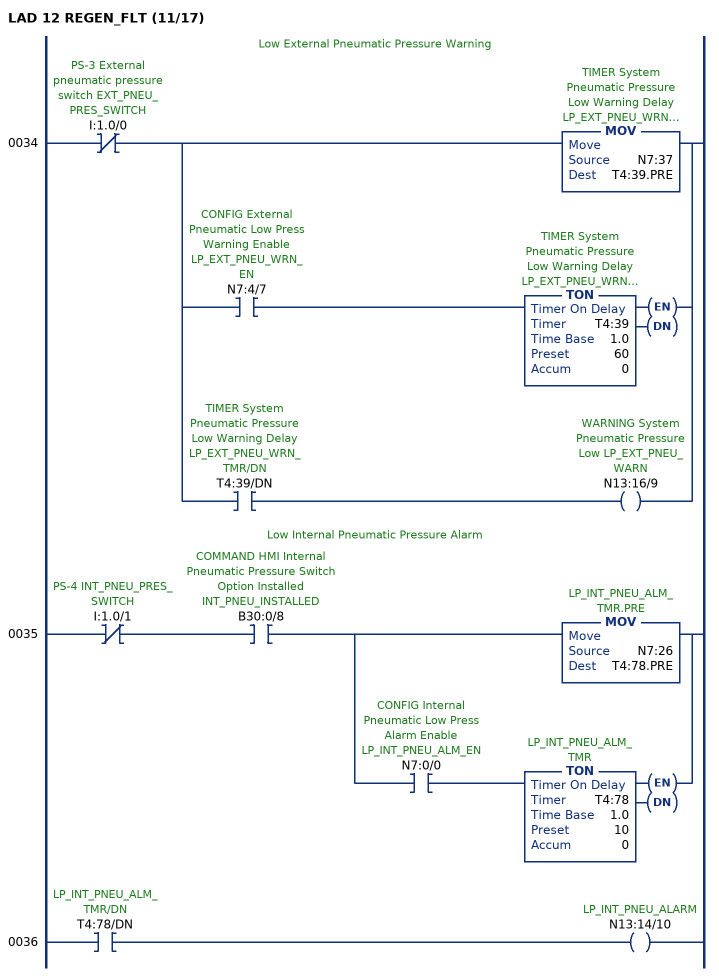
% Rung: 34 %
% Low External Pneumatic Pressure Warning %
SOR XIO I:1.0/0 BST MOV N7:37 T4:39.PRE NXB XIC N7:4/7 TON T4:39 1.0 60 0 NXB XIC T4:39/DN OTE N13:16/9 BND EOR
%   I:1.0/0  EXT_PNEU_PRES_SWITCH  "PS-3 External pneumatic pressure switch" %
%   N7:37  LP_EXT_PNEU_WRN_DLY  "CONFIG External Pneumatic Low Press Warning Delay" %
%   T4:39  LP_EXT_PNEU_WRN_TMR  "TIMER System Pneumatic Pressure Low Warning Delay" %
%   N7:4/7  LP_EXT_PNEU_WRN_EN  "CONFIG External Pneumatic Low Press Warning Enable" %
%   N13:16/9  LP_EXT_PNEU_WARN  "WARNING System Pneumatic Pressure Low" %
% Rung: 35 %
% Low Internal Pneumatic Pressure Alarm %
SOR XIO I:1.0/1 XIC B30:0/8 BST MOV N7:26 T4:78.PRE NXB XIC N7:0/0 TON T4:78 1.0 10 0 BND EOR
%   I:1.0/1  INT_PNEU_PRES_SWITCH  "PS-4" %
%   B30:0/8  INT_PNEU_INSTALLED  "COMMAND HMI Internal Pneumatic Pressure Switch Option Installed" %
%   N7:26  LP_INT_PNEU_ALM_DLY  "CONFIG Internal Pneumatic Low Press Alarm Delay" %
%   T4:78  LP_INT_PNEU_ALM_TMR %
%   N7:0/0  LP_INT_PNEU_ALM_EN  "CONFIG Internal Pneumatic Low Press Alarm Enable" %
% Rung: 36 %
SOR XIC T4:78/DN OTE N13:14/10 EOR
%   T4:78  LP_INT_PNEU_ALM_TMR %
%   N13:14/10  LP_INT_PNEU_ALARM %

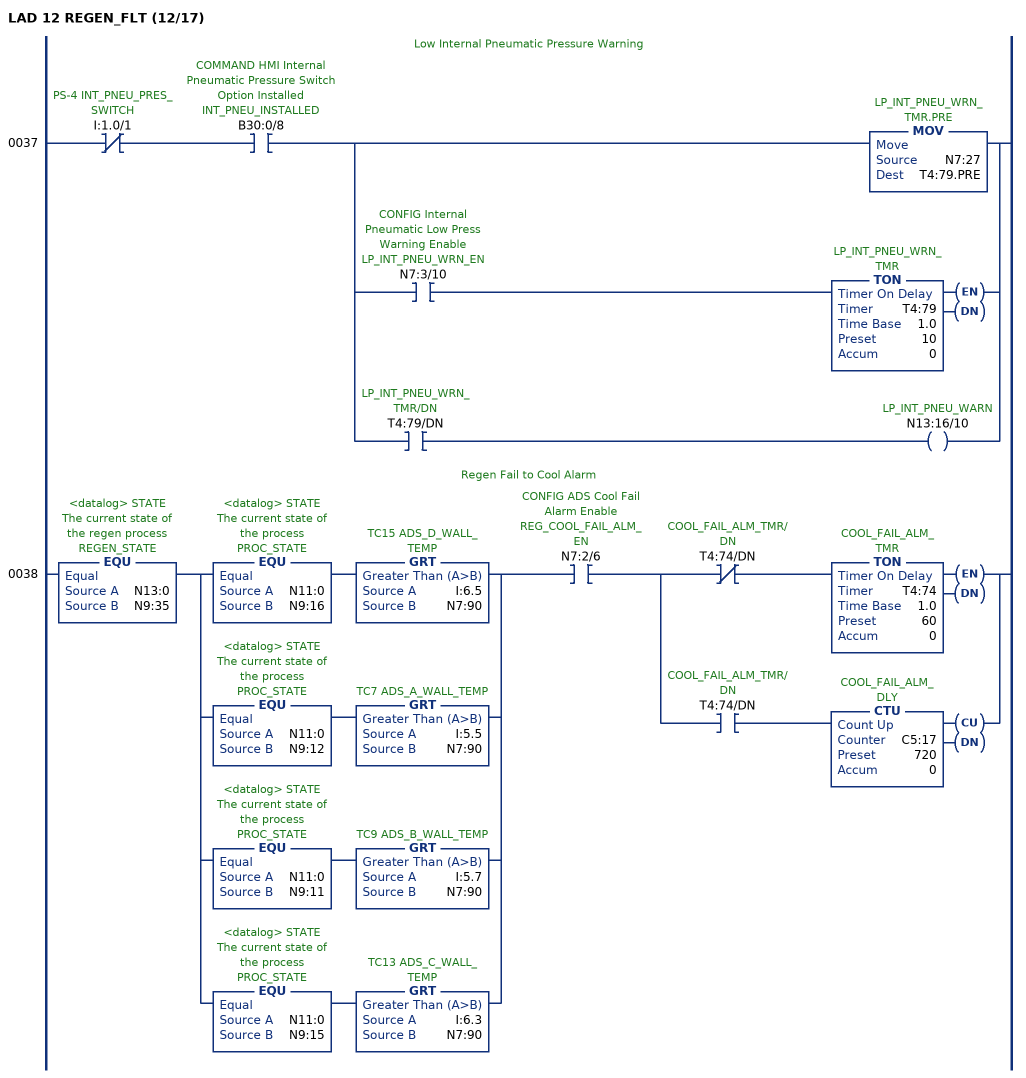
% Rung: 37 %
% Low Internal Pneumatic Pressure Warning %
SOR XIO I:1.0/1 XIC B30:0/8 BST MOV N7:27 T4:79.PRE NXB XIC N7:3/10 TON T4:79 1.0 10 0 NXB XIC T4:79/DN OTE N13:16/10 BND EOR
%   I:1.0/1  INT_PNEU_PRES_SWITCH  "PS-4" %
%   B30:0/8  INT_PNEU_INSTALLED  "COMMAND HMI Internal Pneumatic Pressure Switch Option Installed" %
%   N7:27  LP_INT_PNEU_WRN_DLY  "CONFIG Internal Pneumatic Low Press Warning Delay" %
%   T4:79  LP_INT_PNEU_WRN_TMR %
%   N7:3/10  LP_INT_PNEU_WRN_EN  "CONFIG Internal Pneumatic Low Press Warning Enable" %
%   N13:16/10  LP_INT_PNEU_WARN %
% Rung: 38 %
% Regen Fail to Cool Alarm %
SOR EQU N13:0 N9:35 BST EQU N11:0 N9:16 GRT I:6.5 N7:90 NXB EQU N11:0 N9:12 GRT I:5.5 N7:90 NXB EQU N11:0 N9:11 GRT I:5.7 N7:90 NXB EQU N11:0 N9:15 GRT I:6.3 N7:90 BND XIC N7:2/6 BST XIO T4:74/DN TON T4:74 1.0 60 0 NXB XIC T4:74/DN CTU C5:17 720 0 BND EOR
%   N13:0  REGEN_STATE  "<datalog> STATE The current state of the regen process" %
%   N9:35  REGEN_COOL_WALL  "STATE Regen Cool wall" %
%   N11:0  PROC_STATE  "<datalog> STATE The current state of the process" %
%   N9:16  PROC_REGEN_D  "STATE Process Regen D" %
%   I:6.5  ADS_D_WALL_TEMP  "TC15" %
%   N7:90  REG_COOL_FAIL_ALM_SP  "CONFIG ADS Cool Fail Alarm Setpoint" %
%   N9:12  PROC_REGEN_A  "STATE Process Regen A" %
%   I:5.5  ADS_A_WALL_TEMP  "TC7" %
%   N9:11  PROC_REGEN_B  "STATE Process Regen B" %
%   I:5.7  ADS_B_WALL_TEMP  "TC9" %
%   N9:15  PROC_REGEN_C  "STATE Process Regen C" %
%   I:6.3  ADS_C_WALL_TEMP  "TC13" %
%   N7:2/6  REG_COOL_FAIL_ALM_EN  "CONFIG ADS Cool Fail Alarm Enable" %
%   T4:74  COOL_FAIL_ALM_TMR %
%   C5:17  COOL_FAIL_ALM_DLY %

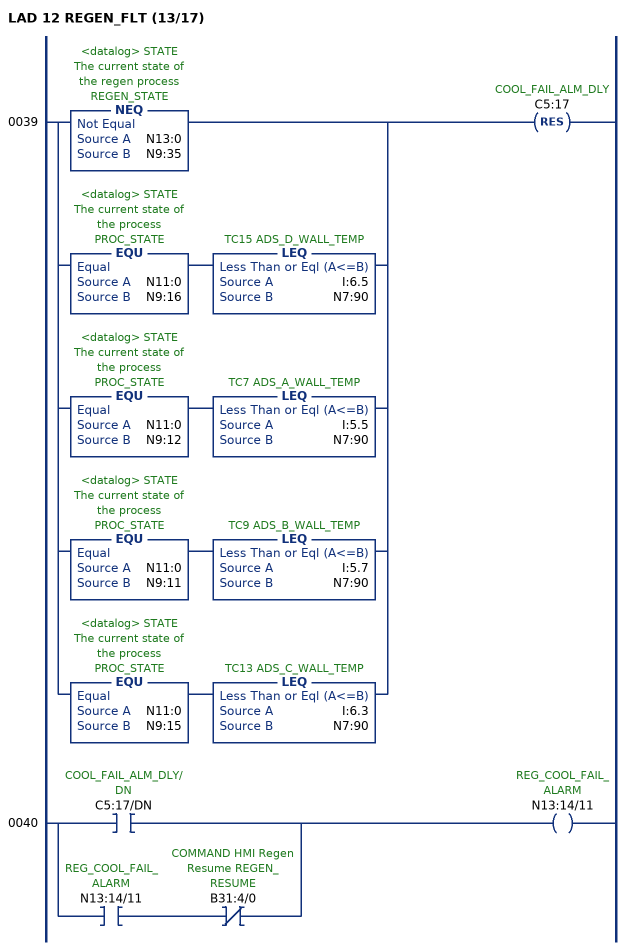
% Rung: 39 %
SOR BST NEQ N13:0 N9:35 NXB EQU N11:0 N9:16 LEQ I:6.5 N7:90 NXB EQU N11:0 N9:12 LEQ I:5.5 N7:90 NXB EQU N11:0 N9:11 LEQ I:5.7 N7:90 NXB EQU N11:0 N9:15 LEQ I:6.3 N7:90 BND RES C5:17 EOR
%   N13:0  REGEN_STATE  "<datalog> STATE The current state of the regen process" %
%   N9:35  REGEN_COOL_WALL  "STATE Regen Cool wall" %
%   N11:0  PROC_STATE  "<datalog> STATE The current state of the process" %
%   N9:16  PROC_REGEN_D  "STATE Process Regen D" %
%   I:6.5  ADS_D_WALL_TEMP  "TC15" %
%   N7:90  REG_COOL_FAIL_ALM_SP  "CONFIG ADS Cool Fail Alarm Setpoint" %
%   N9:12  PROC_REGEN_A  "STATE Process Regen A" %
%   I:5.5  ADS_A_WALL_TEMP  "TC7" %
%   N9:11  PROC_REGEN_B  "STATE Process Regen B" %
%   I:5.7  ADS_B_WALL_TEMP  "TC9" %
%   N9:15  PROC_REGEN_C  "STATE Process Regen C" %
%   I:6.3  ADS_C_WALL_TEMP  "TC13" %
%   C5:17  COOL_FAIL_ALM_DLY %
% Rung: 40 %
SOR BST XIC C5:17/DN NXB XIC N13:14/11 XIO B31:4/0 BND OTE N13:14/11 EOR
%   C5:17  COOL_FAIL_ALM_DLY %
%   N13:14/11  REG_COOL_FAIL_ALARM %
%   B31:4/0  REGEN_RESUME  "COMMAND HMI Regen Resume" %

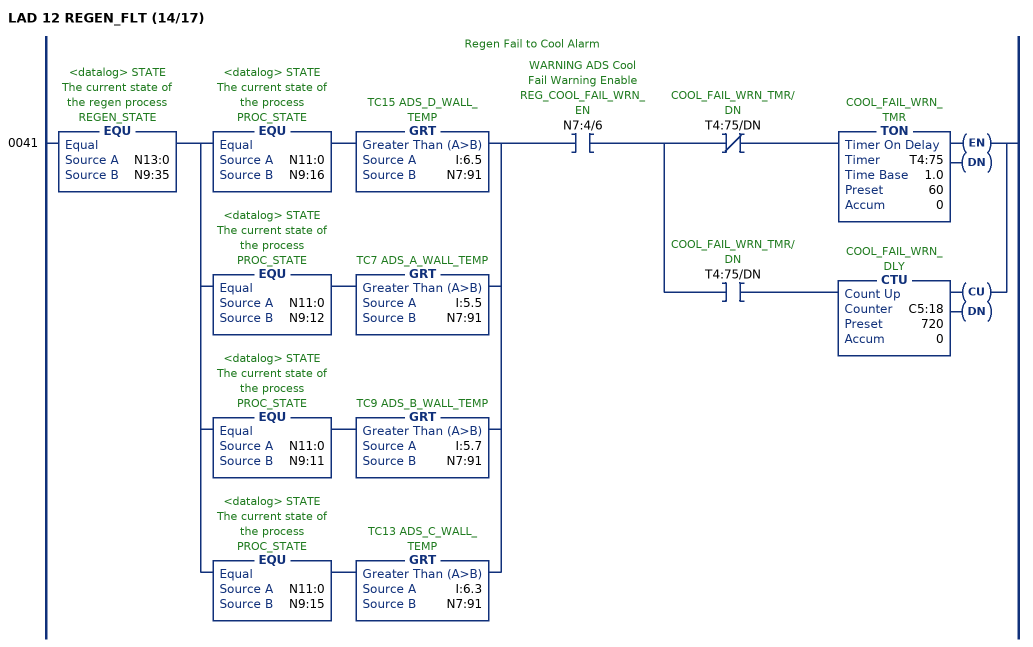
% Rung: 41 %
% Regen Fail to Cool Alarm %
SOR EQU N13:0 N9:35 BST EQU N11:0 N9:16 GRT I:6.5 N7:91 NXB EQU N11:0 N9:12 GRT I:5.5 N7:91 NXB EQU N11:0 N9:11 GRT I:5.7 N7:91 NXB EQU N11:0 N9:15 GRT I:6.3 N7:91 BND XIC N7:4/6 BST XIO T4:75/DN TON T4:75 1.0 60 0 NXB XIC T4:75/DN CTU C5:18 720 0 BND EOR
%   N13:0  REGEN_STATE  "<datalog> STATE The current state of the regen process" %
%   N9:35  REGEN_COOL_WALL  "STATE Regen Cool wall" %
%   N11:0  PROC_STATE  "<datalog> STATE The current state of the process" %
%   N9:16  PROC_REGEN_D  "STATE Process Regen D" %
%   I:6.5  ADS_D_WALL_TEMP  "TC15" %
%   N7:91  REG_COOL_FAIL_WRN_SP  "CONFIG ADS Cool Fail Warning Setpoint" %
%   N9:12  PROC_REGEN_A  "STATE Process Regen A" %
%   I:5.5  ADS_A_WALL_TEMP  "TC7" %
%   N9:11  PROC_REGEN_B  "STATE Process Regen B" %
%   I:5.7  ADS_B_WALL_TEMP  "TC9" %
%   N9:15  PROC_REGEN_C  "STATE Process Regen C" %
%   I:6.3  ADS_C_WALL_TEMP  "TC13" %
%   N7:4/6  REG_COOL_FAIL_WRN_EN  "WARNING ADS Cool Fail Warning Enable" %
%   T4:75  COOL_FAIL_WRN_TMR %
%   C5:18  COOL_FAIL_WRN_DLY %

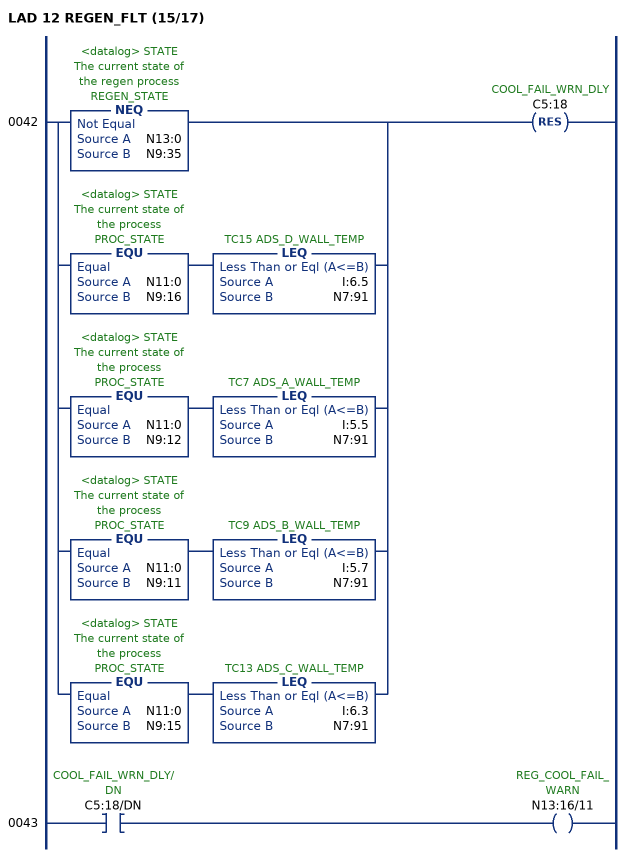
% Rung: 42 %
SOR BST NEQ N13:0 N9:35 NXB EQU N11:0 N9:16 LEQ I:6.5 N7:91 NXB EQU N11:0 N9:12 LEQ I:5.5 N7:91 NXB EQU N11:0 N9:11 LEQ I:5.7 N7:91 NXB EQU N11:0 N9:15 LEQ I:6.3 N7:91 BND RES C5:18 EOR
%   N13:0  REGEN_STATE  "<datalog> STATE The current state of the regen process" %
%   N9:35  REGEN_COOL_WALL  "STATE Regen Cool wall" %
%   N11:0  PROC_STATE  "<datalog> STATE The current state of the process" %
%   N9:16  PROC_REGEN_D  "STATE Process Regen D" %
%   I:6.5  ADS_D_WALL_TEMP  "TC15" %
%   N7:91  REG_COOL_FAIL_WRN_SP  "CONFIG ADS Cool Fail Warning Setpoint" %
%   N9:12  PROC_REGEN_A  "STATE Process Regen A" %
%   I:5.5  ADS_A_WALL_TEMP  "TC7" %
%   N9:11  PROC_REGEN_B  "STATE Process Regen B" %
%   I:5.7  ADS_B_WALL_TEMP  "TC9" %
%   N9:15  PROC_REGEN_C  "STATE Process Regen C" %
%   I:6.3  ADS_C_WALL_TEMP  "TC13" %
%   C5:18  COOL_FAIL_WRN_DLY %
% Rung: 43 %
SOR XIC C5:18/DN OTE N13:16/11 EOR
%   C5:18  COOL_FAIL_WRN_DLY %
%   N13:16/11  REG_COOL_FAIL_WARN %

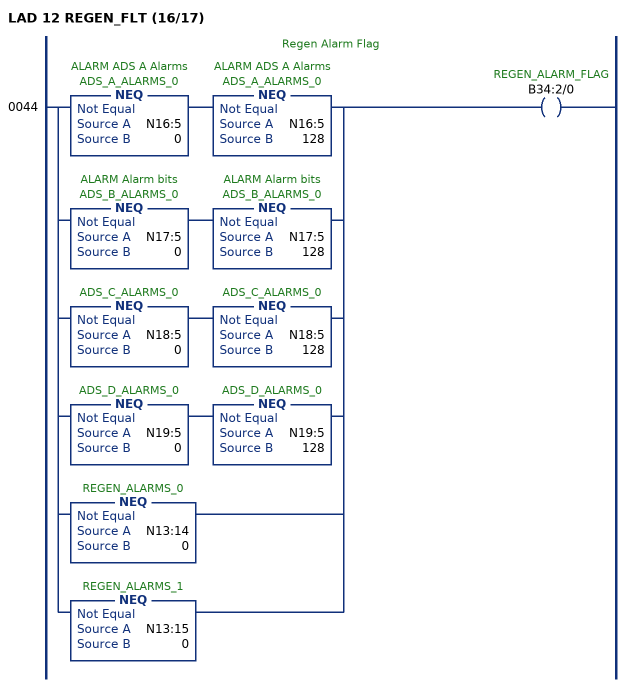
% Rung: 44 %
% Regen Alarm Flag %
SOR BST NEQ N16:5 0 NEQ N16:5 128 NXB NEQ N17:5 0 NEQ N17:5 128 NXB NEQ N18:5 0 NEQ N18:5 128 NXB NEQ N19:5 0 NEQ N19:5 128 NXB NEQ N13:14 0 NXB NEQ N13:15 0 BND OTE B34:2/0 EOR
%   N16:5  ADS_A_ALARMS_0  "ALARM ADS A Alarms" %
%   N17:5  ADS_B_ALARMS_0  "ALARM Alarm bits" %
%   N18:5  ADS_C_ALARMS_0 %
%   N19:5  ADS_D_ALARMS_0 %
%   N13:14  REGEN_ALARMS_0 %
%   N13:15  REGEN_ALARMS_1 %
%   B34:2/0  REGEN_ALARM_FLAG %

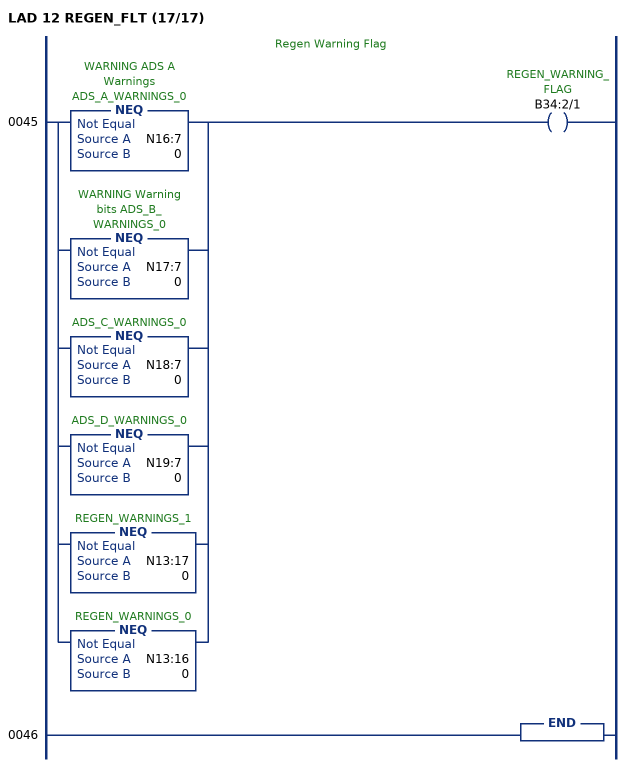
% Rung: 45 %
% Regen Warning Flag %
SOR BST NEQ N16:7 0 NXB NEQ N17:7 0 NXB NEQ N18:7 0 NXB NEQ N19:7 0 NXB NEQ N13:17 0 NXB NEQ N13:16 0 BND OTE B34:2/1 EOR
%   N16:7  ADS_A_WARNINGS_0  "WARNING ADS A Warnings" %
%   N17:7  ADS_B_WARNINGS_0  "WARNING Warning bits" %
%   N18:7  ADS_C_WARNINGS_0 %
%   N19:7  ADS_D_WARNINGS_0 %
%   N13:17  REGEN_WARNINGS_1 %
%   N13:16  REGEN_WARNINGS_0 %
%   B34:2/1  REGEN_WARNING_FLAG %
% Rung: 46 %
SOR END EOR

LADDER 17 "BYPASS"    % Controls the bypass %
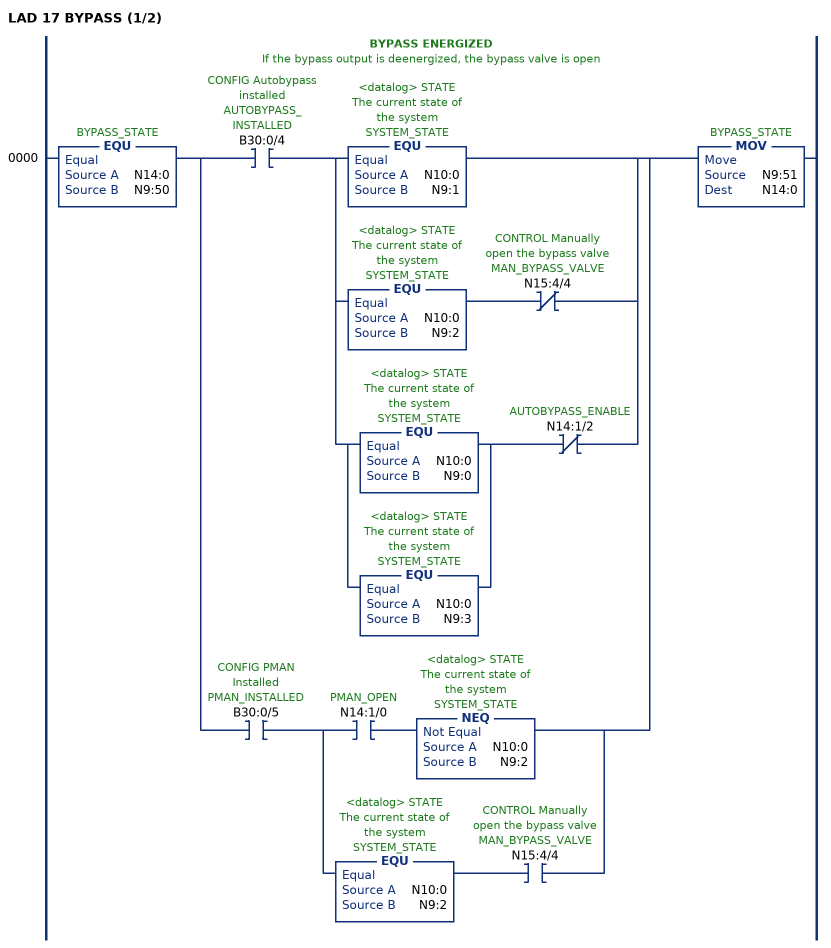
% Rung: 0 %
% TITLE: BYPASS ENERGIZED %
% If the bypass output is deenergized, the bypass valve is open %
SOR EQU N14:0 N9:50 BST XIC B30:0/4 BST EQU N10:0 N9:1 NXB EQU N10:0 N9:2 XIO N15:4/4 NXB BST EQU N10:0 N9:0 NXB EQU N10:0 N9:3 BND XIO N14:1/2 BND NXB XIC B30:0/5 BST XIC N14:1/0 NEQ N10:0 N9:2 NXB EQU N10:0 N9:2 XIC N15:4/4 BND BND MOV N9:51 N14:0 EOR
%   N14:0  BYPASS_STATE %
%   N9:50  BYPASS_DEENERGIZED  "STATE Bypass Deenergized" %
%   B30:0/4  AUTOBYPASS_INSTALLED  "CONFIG Autobypass installed" %
%   N10:0  SYSTEM_STATE  "<datalog> STATE The current state of the system" %
%   N9:1  SYSTEM_PROCESS  "STATE System Process" %
%   N9:2  SYSTEM_MANUAL  "STATE System Manual" %
%   N15:4/4  MAN_BYPASS_VALVE  "CONTROL Manually open the bypass valve" %
%   N9:0  SYSTEM_STANDBY  "STATE System Standby" %
%   N9:3  SYSTEM_ALARM  "STATE System Alarm" %
%   N14:1/2  AUTOBYPASS_ENABLE %
%   B30:0/5  PMAN_INSTALLED  "CONFIG PMAN Installed" %
%   N14:1/0  PMAN_OPEN %
%   N9:51  BYPASS_ENERGIZED  "STATE Bypass Energized" %

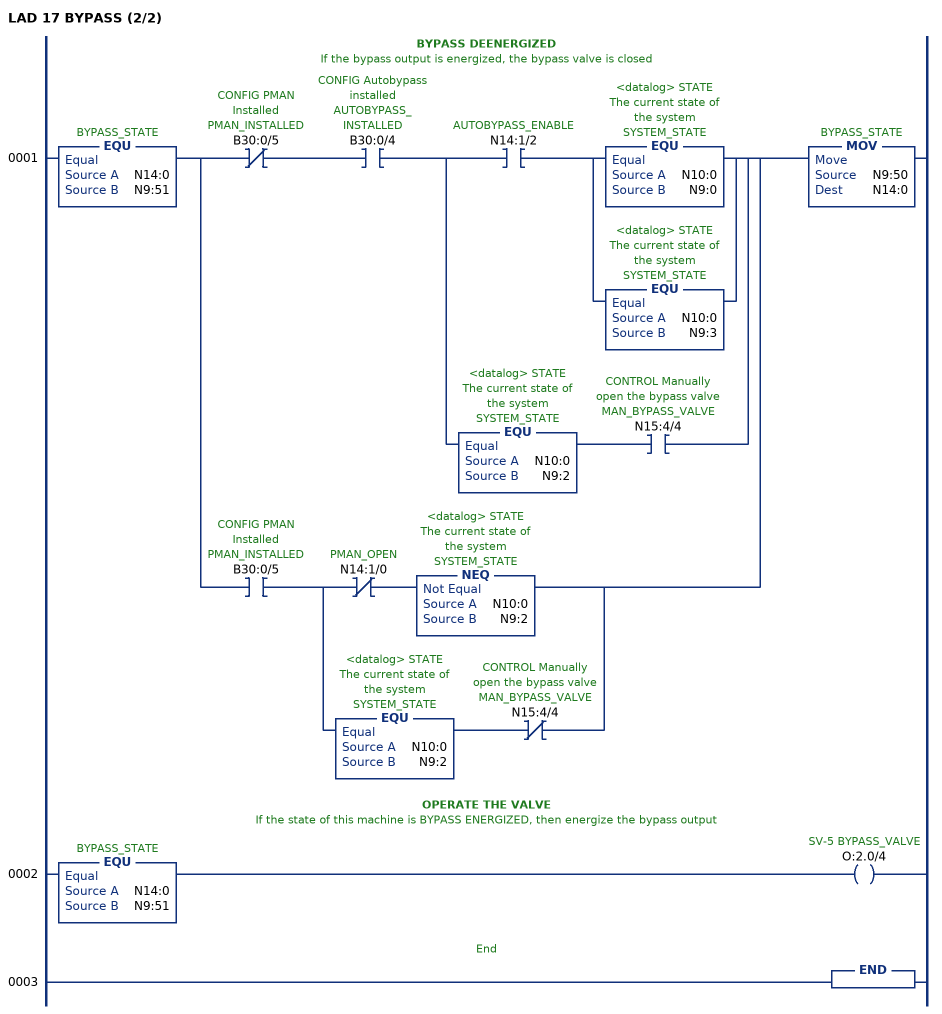
% Rung: 1 %
% TITLE: BYPASS DEENERGIZED %
% If the bypass output is energized, the bypass valve is closed %
SOR EQU N14:0 N9:51 BST XIO B30:0/5 XIC B30:0/4 BST XIC N14:1/2 BST EQU N10:0 N9:0 NXB EQU N10:0 N9:3 BND NXB EQU N10:0 N9:2 XIC N15:4/4 BND NXB XIC B30:0/5 BST XIO N14:1/0 NEQ N10:0 N9:2 NXB EQU N10:0 N9:2 XIO N15:4/4 BND BND MOV N9:50 N14:0 EOR
%   N14:0  BYPASS_STATE %
%   N9:51  BYPASS_ENERGIZED  "STATE Bypass Energized" %
%   B30:0/5  PMAN_INSTALLED  "CONFIG PMAN Installed" %
%   B30:0/4  AUTOBYPASS_INSTALLED  "CONFIG Autobypass installed" %
%   N14:1/2  AUTOBYPASS_ENABLE %
%   N10:0  SYSTEM_STATE  "<datalog> STATE The current state of the system" %
%   N9:0  SYSTEM_STANDBY  "STATE System Standby" %
%   N9:3  SYSTEM_ALARM  "STATE System Alarm" %
%   N9:2  SYSTEM_MANUAL  "STATE System Manual" %
%   N15:4/4  MAN_BYPASS_VALVE  "CONTROL Manually open the bypass valve" %
%   N14:1/0  PMAN_OPEN %
%   N9:50  BYPASS_DEENERGIZED  "STATE Bypass Deenergized" %
% Rung: 2 %
% TITLE: OPERATE THE VALVE %
% If the state of this machine is BYPASS ENERGIZED, then energize the bypass output %
SOR EQU N14:0 N9:51 OTE O:2.0/4 EOR
%   N14:0  BYPASS_STATE %
%   N9:51  BYPASS_ENERGIZED  "STATE Bypass Energized" %
%   O:2.0/4  BYPASS_VALVE  "SV-5" %
% Rung: 3 %
% End %
SOR END EOR

LADDER 18 "MIX PANEL"
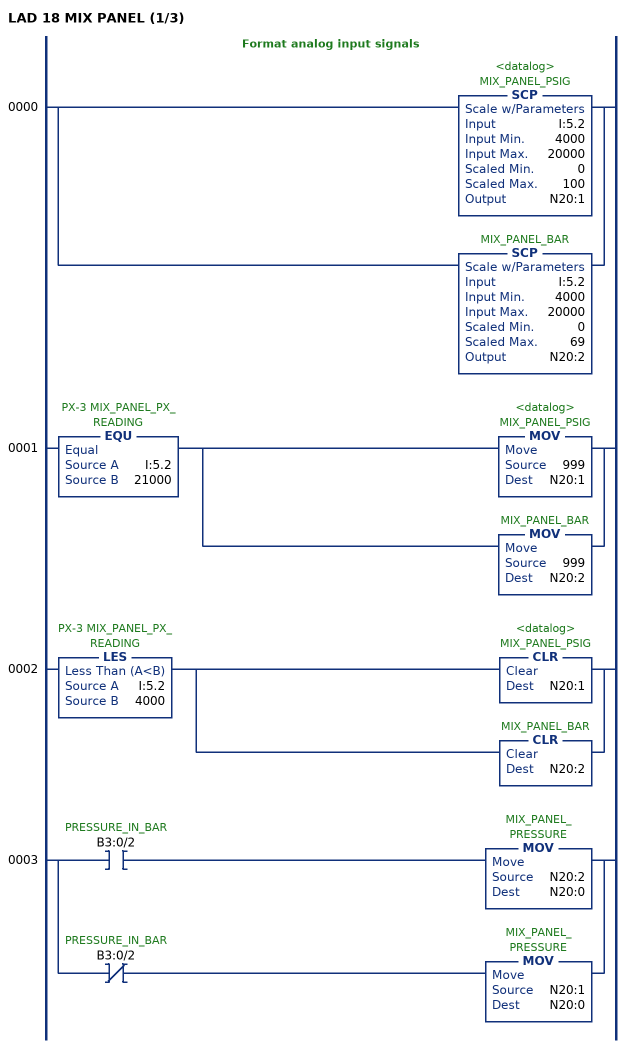
% Rung: 0 %
% TITLE: Format analog input signals %
SOR BST SCP I:5.2 4000 20000 0 100 N20:1 NXB SCP I:5.2 4000 20000 0 69 N20:2 BND EOR
%   I:5.2  MIX_PANEL_PX_READING  "PX-3" %
%   N20:1  MIX_PANEL_PSIG  "<datalog>" %
%   N20:2  MIX_PANEL_BAR %
% Rung: 1 %
SOR EQU I:5.2 21000 BST MOV 999 N20:1 NXB MOV 999 N20:2 BND EOR
%   I:5.2  MIX_PANEL_PX_READING  "PX-3" %
%   N20:1  MIX_PANEL_PSIG  "<datalog>" %
%   N20:2  MIX_PANEL_BAR %
% Rung: 2 %
SOR LES I:5.2 4000 BST CLR N20:1 NXB CLR N20:2 BND EOR
%   I:5.2  MIX_PANEL_PX_READING  "PX-3" %
%   N20:1  MIX_PANEL_PSIG  "<datalog>" %
%   N20:2  MIX_PANEL_BAR %
% Rung: 3 %
SOR BST XIC B3:0/2 MOV N20:2 N20:0 NXB XIO B3:0/2 MOV N20:1 N20:0 BND EOR
%   B3:0/2  PRESSURE_IN_BAR %
%   N20:2  MIX_PANEL_BAR %
%   N20:0  MIX_PANEL_PRESSURE %
%   N20:1  MIX_PANEL_PSIG  "<datalog>" %

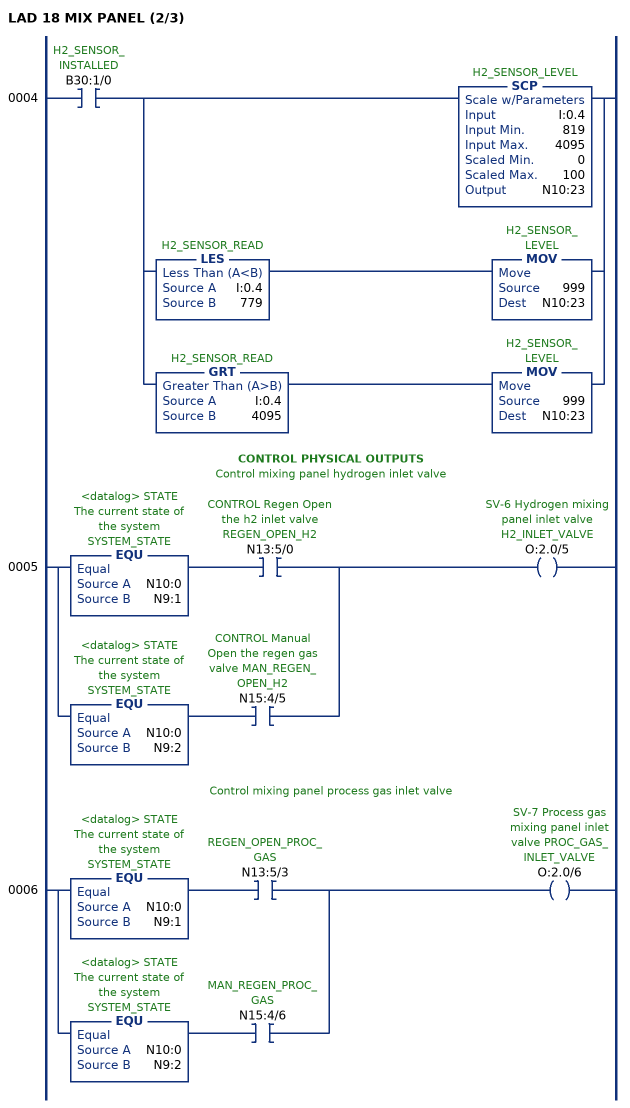
% Rung: 4 %
SOR XIC B30:1/0 BST SCP I:0.4 819 4095 0 100 N10:23 NXB LES I:0.4 779 MOV 999 N10:23 NXB GRT I:0.4 4095 MOV 999 N10:23 BND EOR
%   B30:1/0  H2_SENSOR_INSTALLED %
%   I:0.4  H2_SENSOR_READ %
%   N10:23  H2_SENSOR_LEVEL %
% Rung: 5 %
% TITLE: CONTROL PHYSICAL OUTPUTS %
% Control mixing panel hydrogen inlet valve %
SOR BST EQU N10:0 N9:1 XIC N13:5/0 NXB EQU N10:0 N9:2 XIC N15:4/5 BND OTE O:2.0/5 EOR
%   N10:0  SYSTEM_STATE  "<datalog> STATE The current state of the system" %
%   N9:1  SYSTEM_PROCESS  "STATE System Process" %
%   N13:5/0  REGEN_OPEN_H2  "CONTROL Regen Open the h2 inlet valve" %
%   N9:2  SYSTEM_MANUAL  "STATE System Manual" %
%   N15:4/5  MAN_REGEN_OPEN_H2  "CONTROL Manual Open the regen gas valve" %
%   O:2.0/5  H2_INLET_VALVE  "SV-6 Hydrogen mixing panel inlet valve" %
% Rung: 6 %
% Control mixing panel process gas inlet valve %
SOR BST EQU N10:0 N9:1 XIC N13:5/3 NXB EQU N10:0 N9:2 XIC N15:4/6 BND OTE O:2.0/6 EOR
%   N10:0  SYSTEM_STATE  "<datalog> STATE The current state of the system" %
%   N9:1  SYSTEM_PROCESS  "STATE System Process" %
%   N13:5/3  REGEN_OPEN_PROC_GAS %
%   N9:2  SYSTEM_MANUAL  "STATE System Manual" %
%   N15:4/6  MAN_REGEN_PROC_GAS %
%   O:2.0/6  PROC_GAS_INLET_VALVE  "SV-7 Process gas mixing panel inlet valve" %

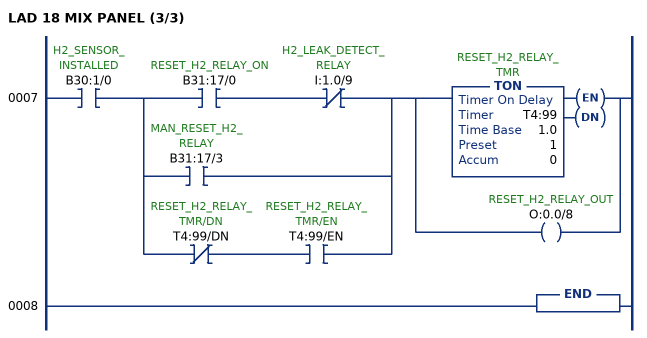
% Rung: 7 %
SOR XIC B30:1/0 BST XIC B31:17/0 XIO I:1.0/9 NXB XIC B31:17/3 NXB XIO T4:99/DN XIC T4:99/EN BND BST TON T4:99 1.0 1 0 NXB OTE O:0.0/8 BND EOR
%   B30:1/0  H2_SENSOR_INSTALLED %
%   B31:17/0  RESET_H2_RELAY_ON %
%   I:1.0/9  H2_LEAK_DETECT_RELAY %
%   B31:17/3  MAN_RESET_H2_RELAY %
%   T4:99  RESET_H2_RELAY_TMR %
%   O:0.0/8  RESET_H2_RELAY_OUT %
% Rung: 8 %
SOR END EOR

LADDER 20 "ADS_A"    % Controls the Adsorber A %
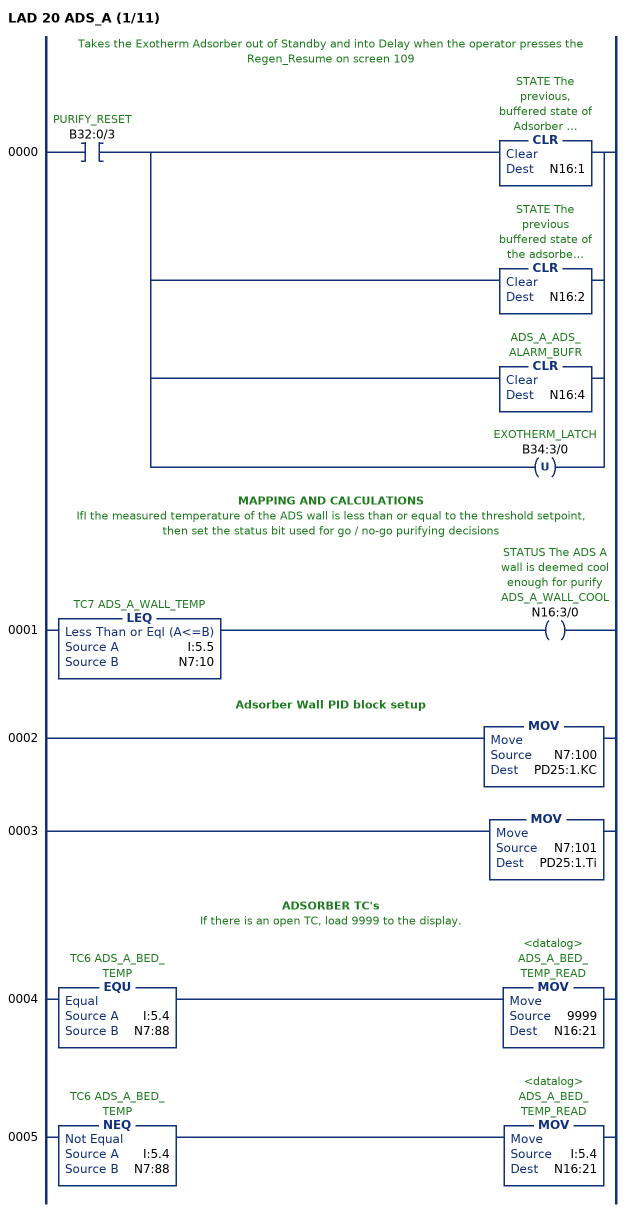
% Rung: 0 %
% Takes the Exotherm Adsorber out of Standby and into Delay when the operator presses the Regen_Resume on screen 109 %
SOR XIC B32:0/3 BST CLR N16:1 NXB CLR N16:2 NXB CLR N16:4 NXB OTU B34:3/0 BND EOR
%   B32:0/3  PURIFY_RESET %
%   N16:1  ADS_A_STANDBY_BUFFER  "STATE The previous, buffered state of Adsorber A" %
%   N16:2  ADS_A_SYS_ALARM_BUFR  "STATE The previous buffered state of the adsorber when the alarm occured" %
%   N16:4  ADS_A_ADS_ALARM_BUFR %
%   B34:3/0  EXOTHERM_LATCH %
% Rung: 1 %
% TITLE: MAPPING AND CALCULATIONS %
% IfI the measured temperature of the ADS wall is less than or equal to the threshold setpoint, then set the status bit used for go / no-go purifying decisions %
SOR LEQ I:5.5 N7:10 OTE N16:3/0 EOR
%   I:5.5  ADS_A_WALL_TEMP  "TC7" %
%   N7:10  ADS_WALL_TEMP_COOL  "CONFIG The temp at which the adsorber wall is deemed to be cool enough to purify" %
%   N16:3/0  ADS_A_WALL_COOL  "STATUS The ADS A wall is deemed cool enough for purify" %
% Rung: 2 %
% TITLE: Adsorber Wall PID block setup %
SOR MOV N7:100 PD25:1.KC EOR
%   N7:100  BLANKET_P  "CONFIG Blanket Proportional Gain" %
% Rung: 3 %
SOR MOV N7:101 PD25:1.Ti EOR
%   N7:101  BLANKET_I  "CONFIG Blanket Integral Gain" %
% Rung: 4 %
% TITLE: ADSORBER TC's %
% If there is an open TC, load 9999 to the display. %
SOR EQU I:5.4 N7:88 MOV 9999 N16:21 EOR
%   I:5.4  ADS_A_BED_TEMP  "TC6" %
%   N7:88  TC_OPEN_SP  "CONFIG TC Open Setpoint" %
%   N16:21  ADS_A_BED_TEMP_READ  "<datalog>" %
% Rung: 5 %
SOR NEQ I:5.4 N7:88 MOV I:5.4 N16:21 EOR
%   I:5.4  ADS_A_BED_TEMP  "TC6" %
%   N7:88  TC_OPEN_SP  "CONFIG TC Open Setpoint" %
%   N16:21  ADS_A_BED_TEMP_READ  "<datalog>" %

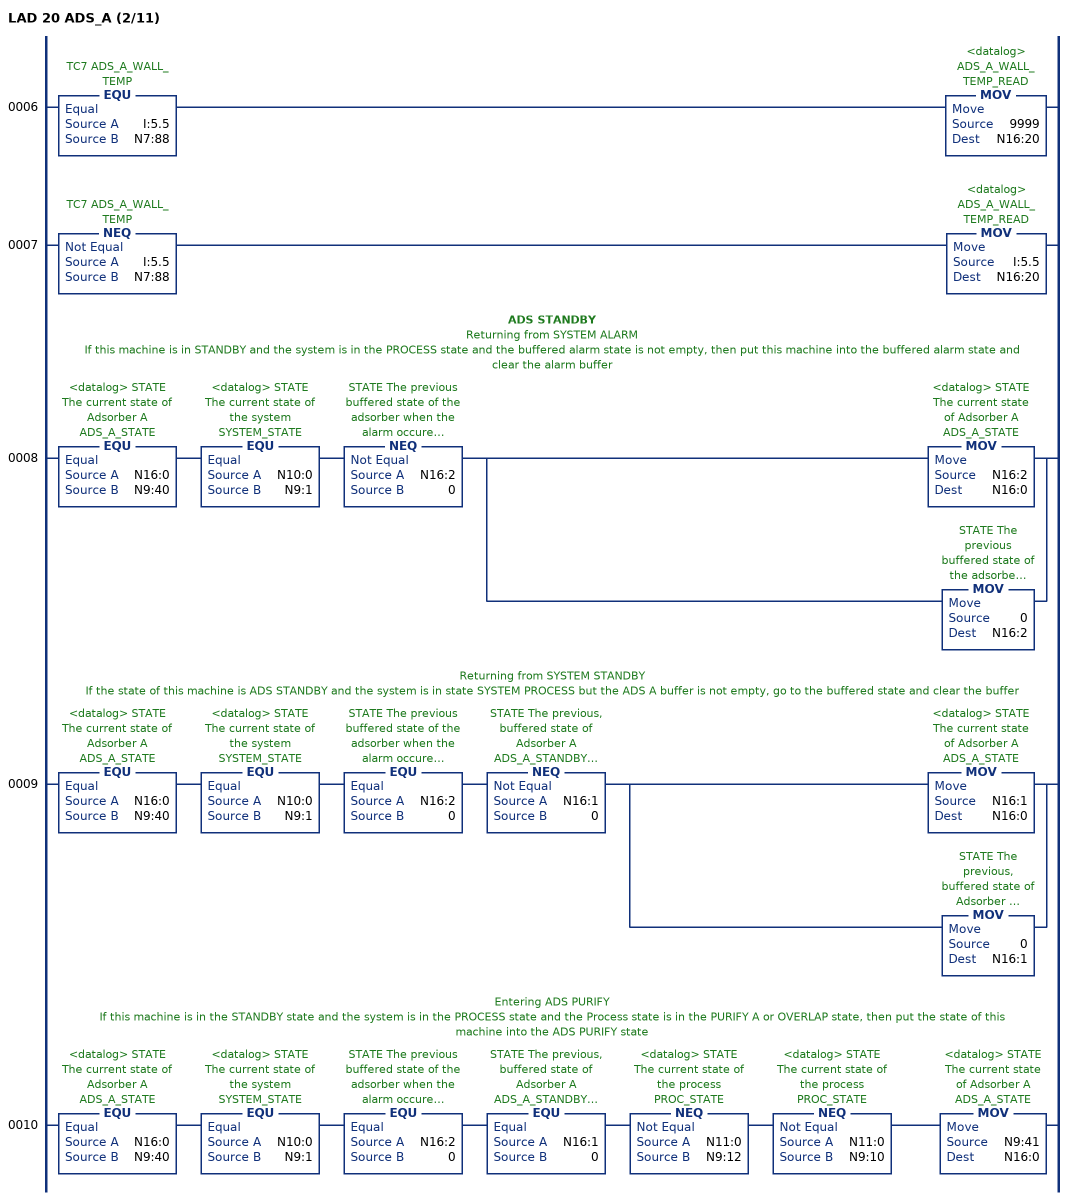
% Rung: 6 %
SOR EQU I:5.5 N7:88 MOV 9999 N16:20 EOR
%   I:5.5  ADS_A_WALL_TEMP  "TC7" %
%   N7:88  TC_OPEN_SP  "CONFIG TC Open Setpoint" %
%   N16:20  ADS_A_WALL_TEMP_READ  "<datalog>" %
% Rung: 7 %
SOR NEQ I:5.5 N7:88 MOV I:5.5 N16:20 EOR
%   I:5.5  ADS_A_WALL_TEMP  "TC7" %
%   N7:88  TC_OPEN_SP  "CONFIG TC Open Setpoint" %
%   N16:20  ADS_A_WALL_TEMP_READ  "<datalog>" %
% Rung: 8 %
% TITLE: ADS STANDBY %
% Returning from SYSTEM ALARM
% If this machine is in STANDBY and the system is in the PROCESS state and the buffered alarm state is not empty, then put this machine into the buffered alarm state and clear the alarm buffer %
SOR EQU N16:0 N9:40 EQU N10:0 N9:1 NEQ N16:2 0 BST MOV N16:2 N16:0 NXB MOV 0 N16:2 BND EOR
%   N16:0  ADS_A_STATE  "<datalog> STATE The current state of Adsorber A" %
%   N9:40  ADS_STANDBY  "STATE ADS Standby" %
%   N10:0  SYSTEM_STATE  "<datalog> STATE The current state of the system" %
%   N9:1  SYSTEM_PROCESS  "STATE System Process" %
%   N16:2  ADS_A_SYS_ALARM_BUFR  "STATE The previous buffered state of the adsorber when the alarm occured" %
% Rung: 9 %
% Returning from SYSTEM STANDBY
% If the state of this machine is ADS STANDBY and the system is in state SYSTEM PROCESS but the ADS A buffer is not empty, go to the buffered state and clear the buffer %
SOR EQU N16:0 N9:40 EQU N10:0 N9:1 EQU N16:2 0 NEQ N16:1 0 BST MOV N16:1 N16:0 NXB MOV 0 N16:1 BND EOR
%   N16:0  ADS_A_STATE  "<datalog> STATE The current state of Adsorber A" %
%   N9:40  ADS_STANDBY  "STATE ADS Standby" %
%   N10:0  SYSTEM_STATE  "<datalog> STATE The current state of the system" %
%   N9:1  SYSTEM_PROCESS  "STATE System Process" %
%   N16:2  ADS_A_SYS_ALARM_BUFR  "STATE The previous buffered state of the adsorber when the alarm occured" %
%   N16:1  ADS_A_STANDBY_BUFFER  "STATE The previous, buffered state of Adsorber A" %
% Rung: 10 %
% Entering ADS PURIFY
% If this machine is in the STANDBY state and the system is in the PROCESS state and the Process state is in the PURIFY A or OVERLAP state, then put the state of this machine into the ADS PURIFY state %
SOR EQU N16:0 N9:40 EQU N10:0 N9:1 EQU N16:2 0 EQU N16:1 0 NEQ N11:0 N9:12 NEQ N11:0 N9:10 MOV N9:41 N16:0 EOR
%   N16:0  ADS_A_STATE  "<datalog> STATE The current state of Adsorber A" %
%   N9:40  ADS_STANDBY  "STATE ADS Standby" %
%   N10:0  SYSTEM_STATE  "<datalog> STATE The current state of the system" %
%   N9:1  SYSTEM_PROCESS  "STATE System Process" %
%   N16:2  ADS_A_SYS_ALARM_BUFR  "STATE The previous buffered state of the adsorber when the alarm occured" %
%   N16:1  ADS_A_STANDBY_BUFFER  "STATE The previous, buffered state of Adsorber A" %
%   N11:0  PROC_STATE  "<datalog> STATE The current state of the process" %
%   N9:12  PROC_REGEN_A  "STATE Process Regen A" %
%   N9:10  PROCESS_STANDBY  "STATE Process Standby" %
%   N9:41  ADS_PURIFY  "STATE ADS Purify" %

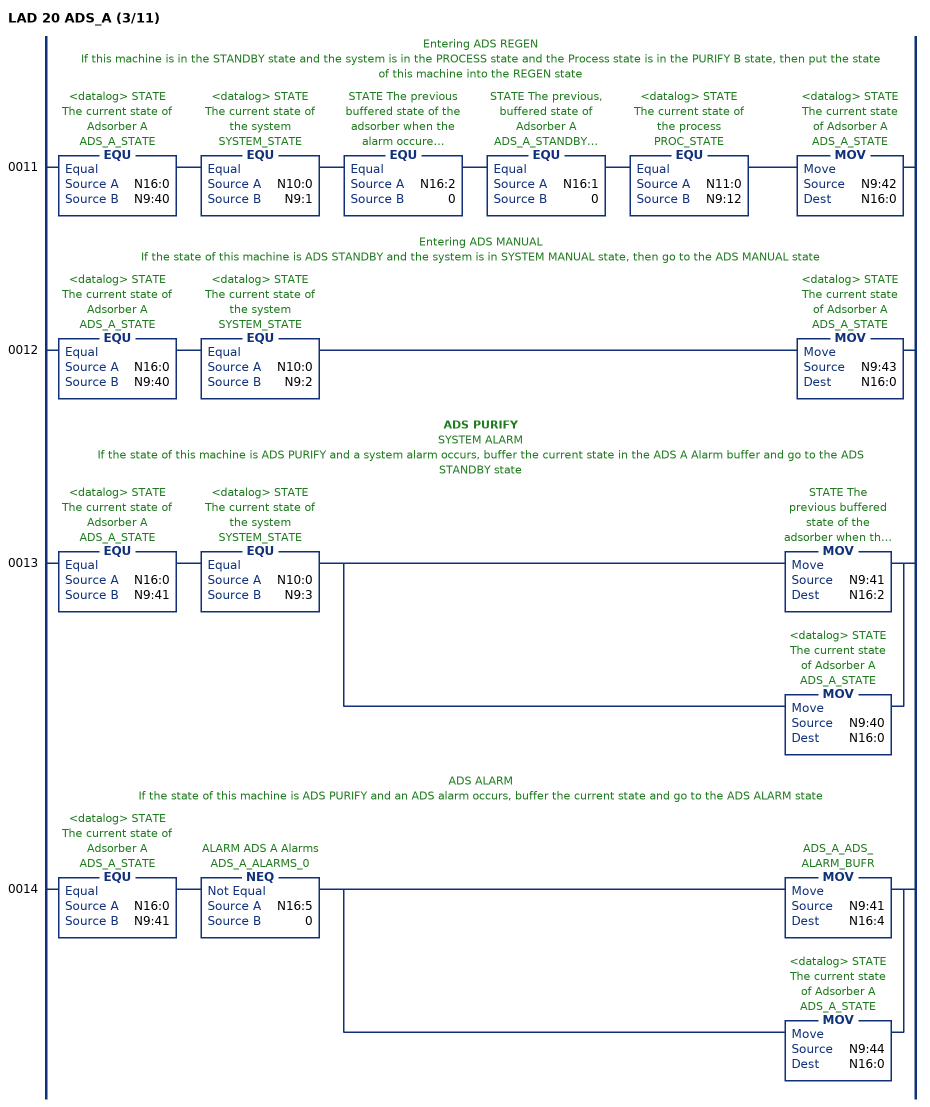
% Rung: 11 %
% Entering ADS REGEN
% If this machine is in the STANDBY state and the system is in the PROCESS state and the Process state is in the PURIFY B state, then put the state of this machine into the REGEN state %
SOR EQU N16:0 N9:40 EQU N10:0 N9:1 EQU N16:2 0 EQU N16:1 0 EQU N11:0 N9:12 MOV N9:42 N16:0 EOR
%   N16:0  ADS_A_STATE  "<datalog> STATE The current state of Adsorber A" %
%   N9:40  ADS_STANDBY  "STATE ADS Standby" %
%   N10:0  SYSTEM_STATE  "<datalog> STATE The current state of the system" %
%   N9:1  SYSTEM_PROCESS  "STATE System Process" %
%   N16:2  ADS_A_SYS_ALARM_BUFR  "STATE The previous buffered state of the adsorber when the alarm occured" %
%   N16:1  ADS_A_STANDBY_BUFFER  "STATE The previous, buffered state of Adsorber A" %
%   N11:0  PROC_STATE  "<datalog> STATE The current state of the process" %
%   N9:12  PROC_REGEN_A  "STATE Process Regen A" %
%   N9:42  ADS_REGEN  "STATE ADS Regen" %
% Rung: 12 %
% Entering ADS MANUAL
% If the state of this machine is ADS STANDBY and the system is in SYSTEM MANUAL state, then go to the ADS MANUAL state %
SOR EQU N16:0 N9:40 EQU N10:0 N9:2 MOV N9:43 N16:0 EOR
%   N16:0  ADS_A_STATE  "<datalog> STATE The current state of Adsorber A" %
%   N9:40  ADS_STANDBY  "STATE ADS Standby" %
%   N10:0  SYSTEM_STATE  "<datalog> STATE The current state of the system" %
%   N9:2  SYSTEM_MANUAL  "STATE System Manual" %
%   N9:43  ADS_MANUAL  "STATE ADS Manual" %
% Rung: 13 %
% TITLE: ADS PURIFY %
% SYSTEM ALARM
% If the state of this machine is ADS PURIFY and a system alarm occurs, buffer the current state in the ADS A Alarm buffer and go to the ADS STANDBY state %
SOR EQU N16:0 N9:41 EQU N10:0 N9:3 BST MOV N9:41 N16:2 NXB MOV N9:40 N16:0 BND EOR
%   N16:0  ADS_A_STATE  "<datalog> STATE The current state of Adsorber A" %
%   N9:41  ADS_PURIFY  "STATE ADS Purify" %
%   N10:0  SYSTEM_STATE  "<datalog> STATE The current state of the system" %
%   N9:3  SYSTEM_ALARM  "STATE System Alarm" %
%   N16:2  ADS_A_SYS_ALARM_BUFR  "STATE The previous buffered state of the adsorber when the alarm occured" %
%   N9:40  ADS_STANDBY  "STATE ADS Standby" %
% Rung: 14 %
% ADS ALARM
% If the state of this machine is ADS PURIFY and an ADS alarm occurs, buffer the current state and go to the ADS ALARM state %
SOR EQU N16:0 N9:41 NEQ N16:5 0 BST MOV N9:41 N16:4 NXB MOV N9:44 N16:0 BND EOR
%   N16:0  ADS_A_STATE  "<datalog> STATE The current state of Adsorber A" %
%   N9:41  ADS_PURIFY  "STATE ADS Purify" %
%   N16:5  ADS_A_ALARMS_0  "ALARM ADS A Alarms" %
%   N16:4  ADS_A_ADS_ALARM_BUFR %
%   N9:44  ADS_ALARM  "STATE ADS Alarm" %

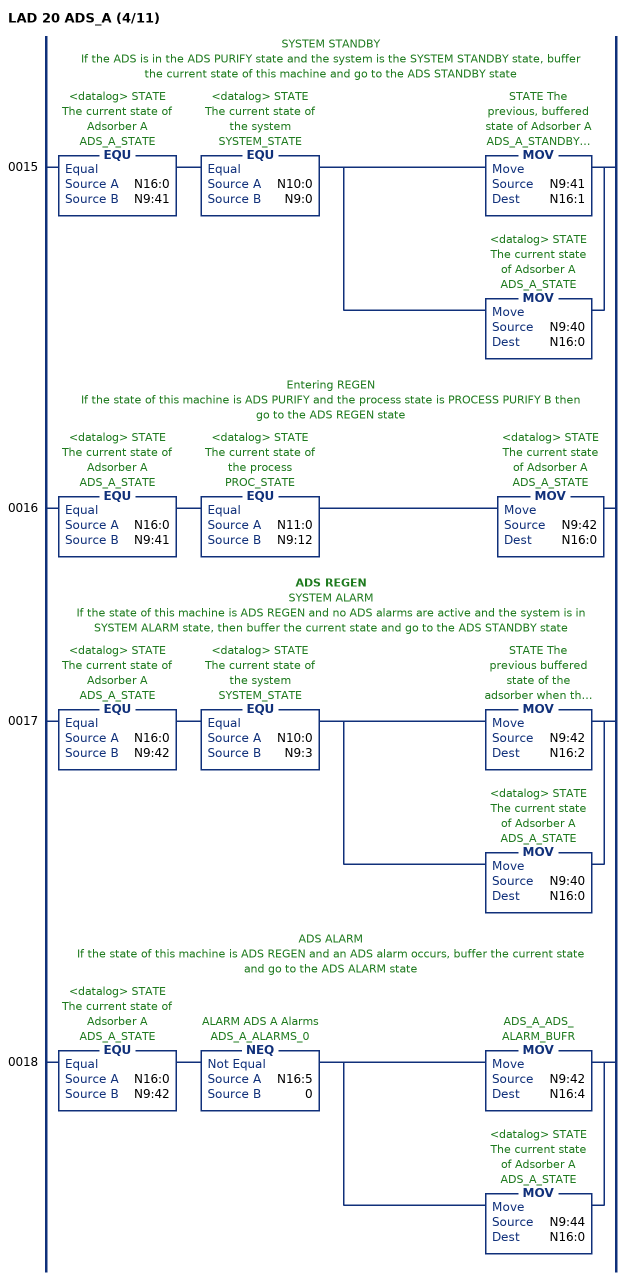
% Rung: 15 %
% SYSTEM STANDBY
% If the ADS is in the ADS PURIFY state and the system is the SYSTEM STANDBY state, buffer the current state of this machine and go to the ADS STANDBY state %
SOR EQU N16:0 N9:41 EQU N10:0 N9:0 BST MOV N9:41 N16:1 NXB MOV N9:40 N16:0 BND EOR
%   N16:0  ADS_A_STATE  "<datalog> STATE The current state of Adsorber A" %
%   N9:41  ADS_PURIFY  "STATE ADS Purify" %
%   N10:0  SYSTEM_STATE  "<datalog> STATE The current state of the system" %
%   N9:0  SYSTEM_STANDBY  "STATE System Standby" %
%   N16:1  ADS_A_STANDBY_BUFFER  "STATE The previous, buffered state of Adsorber A" %
%   N9:40  ADS_STANDBY  "STATE ADS Standby" %
% Rung: 16 %
% Entering REGEN
% If the state of this machine is ADS PURIFY and the process state is PROCESS PURIFY B then go to the ADS REGEN state %
SOR EQU N16:0 N9:41 EQU N11:0 N9:12 MOV N9:42 N16:0 EOR
%   N16:0  ADS_A_STATE  "<datalog> STATE The current state of Adsorber A" %
%   N9:41  ADS_PURIFY  "STATE ADS Purify" %
%   N11:0  PROC_STATE  "<datalog> STATE The current state of the process" %
%   N9:12  PROC_REGEN_A  "STATE Process Regen A" %
%   N9:42  ADS_REGEN  "STATE ADS Regen" %
% Rung: 17 %
% TITLE: ADS REGEN %
% SYSTEM ALARM
% If the state of this machine is ADS REGEN and no ADS alarms are active and the system is in SYSTEM ALARM state, then buffer the current state and go to the ADS STANDBY state %
SOR EQU N16:0 N9:42 EQU N10:0 N9:3 BST MOV N9:42 N16:2 NXB MOV N9:40 N16:0 BND EOR
%   N16:0  ADS_A_STATE  "<datalog> STATE The current state of Adsorber A" %
%   N9:42  ADS_REGEN  "STATE ADS Regen" %
%   N10:0  SYSTEM_STATE  "<datalog> STATE The current state of the system" %
%   N9:3  SYSTEM_ALARM  "STATE System Alarm" %
%   N16:2  ADS_A_SYS_ALARM_BUFR  "STATE The previous buffered state of the adsorber when the alarm occured" %
%   N9:40  ADS_STANDBY  "STATE ADS Standby" %
% Rung: 18 %
% ADS ALARM
% If the state of this machine is ADS REGEN and an ADS alarm occurs, buffer the current state and go to the ADS ALARM state %
SOR EQU N16:0 N9:42 NEQ N16:5 0 BST MOV N9:42 N16:4 NXB MOV N9:44 N16:0 BND EOR
%   N16:0  ADS_A_STATE  "<datalog> STATE The current state of Adsorber A" %
%   N9:42  ADS_REGEN  "STATE ADS Regen" %
%   N16:5  ADS_A_ALARMS_0  "ALARM ADS A Alarms" %
%   N16:4  ADS_A_ADS_ALARM_BUFR %
%   N9:44  ADS_ALARM  "STATE ADS Alarm" %

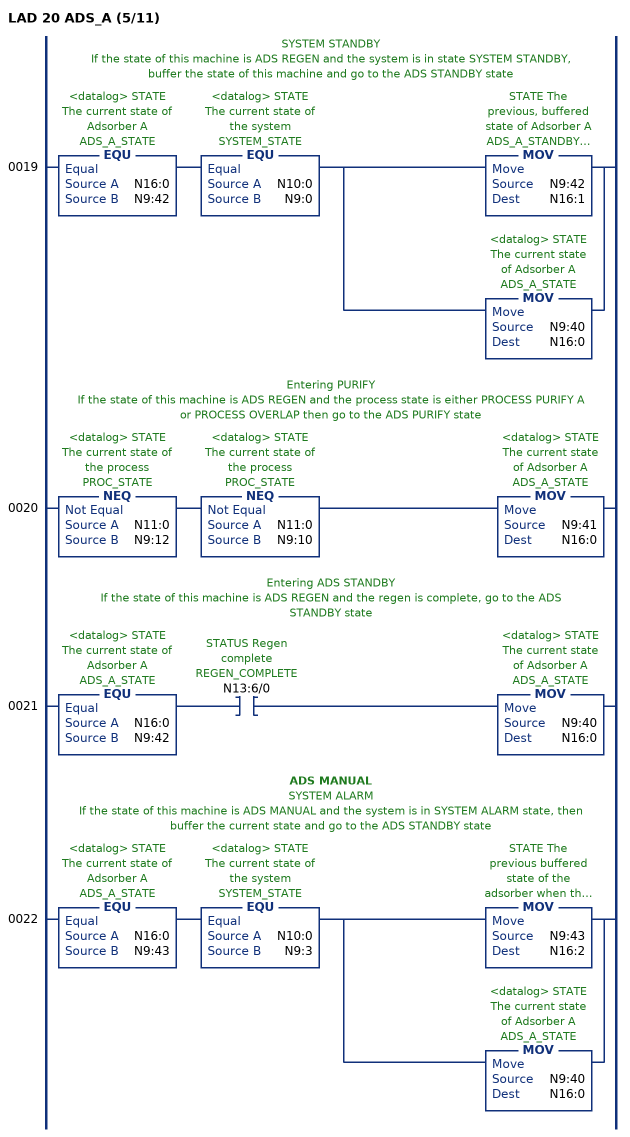
% Rung: 19 %
% SYSTEM STANDBY
% If the state of this machine is ADS REGEN and the system is in state SYSTEM STANDBY, buffer the state of this machine and go to the ADS STANDBY state %
SOR EQU N16:0 N9:42 EQU N10:0 N9:0 BST MOV N9:42 N16:1 NXB MOV N9:40 N16:0 BND EOR
%   N16:0  ADS_A_STATE  "<datalog> STATE The current state of Adsorber A" %
%   N9:42  ADS_REGEN  "STATE ADS Regen" %
%   N10:0  SYSTEM_STATE  "<datalog> STATE The current state of the system" %
%   N9:0  SYSTEM_STANDBY  "STATE System Standby" %
%   N16:1  ADS_A_STANDBY_BUFFER  "STATE The previous, buffered state of Adsorber A" %
%   N9:40  ADS_STANDBY  "STATE ADS Standby" %
% Rung: 20 %
% Entering PURIFY
% If the state of this machine is ADS REGEN and the process state is either PROCESS PURIFY A or PROCESS OVERLAP then go to the ADS PURIFY state %
SOR NEQ N11:0 N9:12 NEQ N11:0 N9:10 MOV N9:41 N16:0 EOR
%   N11:0  PROC_STATE  "<datalog> STATE The current state of the process" %
%   N9:12  PROC_REGEN_A  "STATE Process Regen A" %
%   N9:10  PROCESS_STANDBY  "STATE Process Standby" %
%   N9:41  ADS_PURIFY  "STATE ADS Purify" %
%   N16:0  ADS_A_STATE  "<datalog> STATE The current state of Adsorber A" %
% Rung: 21 %
% Entering ADS STANDBY
% If the state of this machine is ADS REGEN and the regen is complete, go to the ADS STANDBY state %
SOR EQU N16:0 N9:42 XIC N13:6/0 MOV N9:40 N16:0 EOR
%   N16:0  ADS_A_STATE  "<datalog> STATE The current state of Adsorber A" %
%   N9:42  ADS_REGEN  "STATE ADS Regen" %
%   N13:6/0  REGEN_COMPLETE  "STATUS Regen complete" %
%   N9:40  ADS_STANDBY  "STATE ADS Standby" %
% Rung: 22 %
% TITLE: ADS MANUAL %
% SYSTEM ALARM
% If the state of this machine is ADS MANUAL and the system is in SYSTEM ALARM state, then buffer the current state and go to the ADS STANDBY state %
SOR EQU N16:0 N9:43 EQU N10:0 N9:3 BST MOV N9:43 N16:2 NXB MOV N9:40 N16:0 BND EOR
%   N16:0  ADS_A_STATE  "<datalog> STATE The current state of Adsorber A" %
%   N9:43  ADS_MANUAL  "STATE ADS Manual" %
%   N10:0  SYSTEM_STATE  "<datalog> STATE The current state of the system" %
%   N9:3  SYSTEM_ALARM  "STATE System Alarm" %
%   N16:2  ADS_A_SYS_ALARM_BUFR  "STATE The previous buffered state of the adsorber when the alarm occured" %
%   N9:40  ADS_STANDBY  "STATE ADS Standby" %

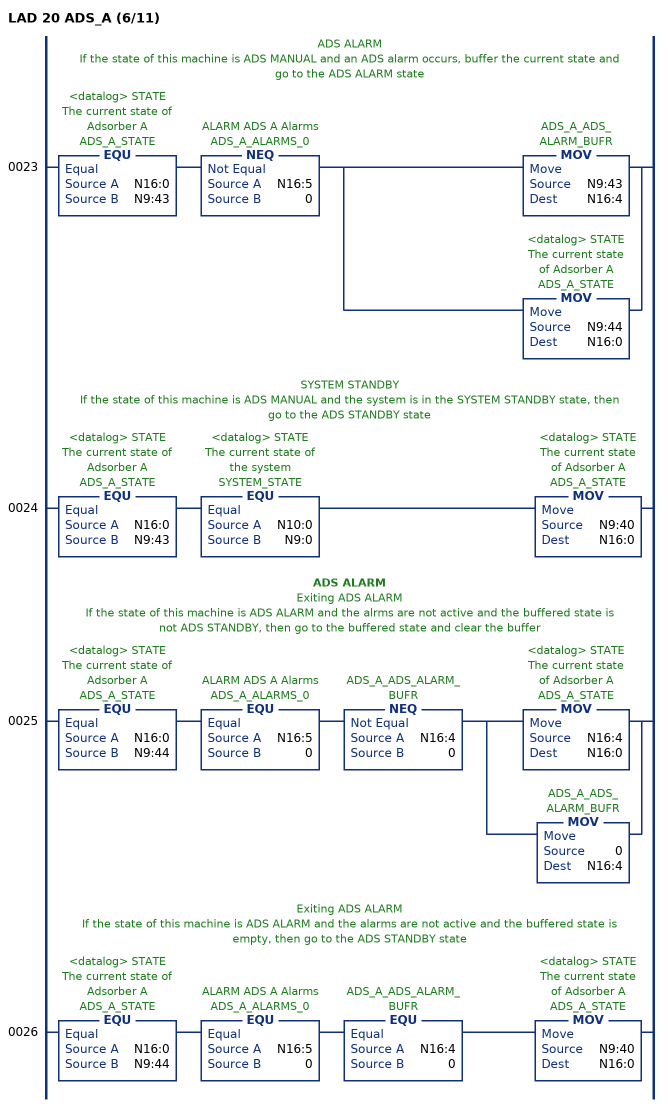
% Rung: 23 %
% ADS ALARM
% If the state of this machine is ADS MANUAL and an ADS alarm occurs, buffer the current state and go to the ADS ALARM state %
SOR EQU N16:0 N9:43 NEQ N16:5 0 BST MOV N9:43 N16:4 NXB MOV N9:44 N16:0 BND EOR
%   N16:0  ADS_A_STATE  "<datalog> STATE The current state of Adsorber A" %
%   N9:43  ADS_MANUAL  "STATE ADS Manual" %
%   N16:5  ADS_A_ALARMS_0  "ALARM ADS A Alarms" %
%   N16:4  ADS_A_ADS_ALARM_BUFR %
%   N9:44  ADS_ALARM  "STATE ADS Alarm" %
% Rung: 24 %
% SYSTEM STANDBY
% If the state of this machine is ADS MANUAL and the system is in the SYSTEM STANDBY state, then go to the ADS STANDBY state %
SOR EQU N16:0 N9:43 EQU N10:0 N9:0 MOV N9:40 N16:0 EOR
%   N16:0  ADS_A_STATE  "<datalog> STATE The current state of Adsorber A" %
%   N9:43  ADS_MANUAL  "STATE ADS Manual" %
%   N10:0  SYSTEM_STATE  "<datalog> STATE The current state of the system" %
%   N9:0  SYSTEM_STANDBY  "STATE System Standby" %
%   N9:40  ADS_STANDBY  "STATE ADS Standby" %
% Rung: 25 %
% TITLE: ADS ALARM %
% Exiting ADS ALARM
% If the state of this machine is ADS ALARM and the alrms are not active and the buffered state is not ADS STANDBY, then go to the buffered state and clear the buffer %
SOR EQU N16:0 N9:44 EQU N16:5 0 NEQ N16:4 0 BST MOV N16:4 N16:0 NXB MOV 0 N16:4 BND EOR
%   N16:0  ADS_A_STATE  "<datalog> STATE The current state of Adsorber A" %
%   N9:44  ADS_ALARM  "STATE ADS Alarm" %
%   N16:5  ADS_A_ALARMS_0  "ALARM ADS A Alarms" %
%   N16:4  ADS_A_ADS_ALARM_BUFR %
% Rung: 26 %
% Exiting ADS ALARM
% If the state of this machine is ADS ALARM and the alarms are not active and the buffered state is empty, then go to the ADS STANDBY state %
SOR EQU N16:0 N9:44 EQU N16:5 0 EQU N16:4 0 MOV N9:40 N16:0 EOR
%   N16:0  ADS_A_STATE  "<datalog> STATE The current state of Adsorber A" %
%   N9:44  ADS_ALARM  "STATE ADS Alarm" %
%   N16:5  ADS_A_ALARMS_0  "ALARM ADS A Alarms" %
%   N16:4  ADS_A_ADS_ALARM_BUFR %
%   N9:40  ADS_STANDBY  "STATE ADS Standby" %

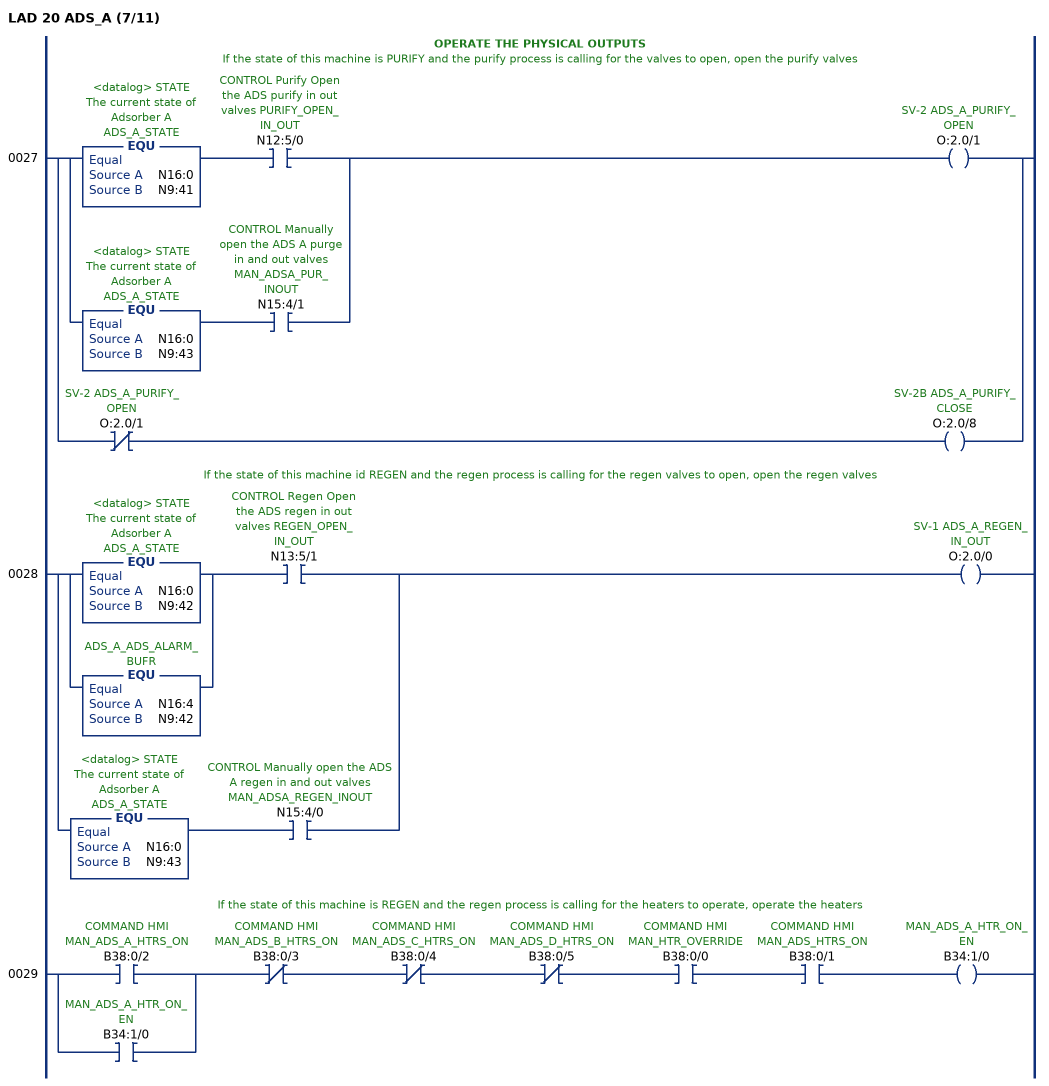
% Rung: 27 %
% TITLE: OPERATE THE PHYSICAL OUTPUTS %
% If the state of this machine is PURIFY and the purify process is calling for the valves to open, open the purify valves %
SOR BST BST EQU N16:0 N9:41 XIC N12:5/0 NXB EQU N16:0 N9:43 XIC N15:4/1 BND OTE O:2.0/1 NXB XIO O:2.0/1 OTE O:2.0/8 BND EOR
%   N16:0  ADS_A_STATE  "<datalog> STATE The current state of Adsorber A" %
%   N9:41  ADS_PURIFY  "STATE ADS Purify" %
%   N12:5/0  PURIFY_OPEN_IN_OUT  "CONTROL Purify Open the ADS purify in out valves" %
%   N9:43  ADS_MANUAL  "STATE ADS Manual" %
%   N15:4/1  MAN_ADSA_PUR_INOUT  "CONTROL Manually open the ADS A purge in and out valves" %
%   O:2.0/1  ADS_A_PURIFY_OPEN  "SV-2" %
%   O:2.0/8  ADS_A_PURIFY_CLOSE  "SV-2B" %
% Rung: 28 %
% If the state of this machine id REGEN and the regen process is calling for the regen valves to open, open the regen valves %
SOR BST BST EQU N16:0 N9:42 NXB EQU N16:4 N9:42 BND XIC N13:5/1 NXB EQU N16:0 N9:43 XIC N15:4/0 BND OTE O:2.0/0 EOR
%   N16:0  ADS_A_STATE  "<datalog> STATE The current state of Adsorber A" %
%   N9:42  ADS_REGEN  "STATE ADS Regen" %
%   N16:4  ADS_A_ADS_ALARM_BUFR %
%   N13:5/1  REGEN_OPEN_IN_OUT  "CONTROL Regen Open the ADS regen in out valves" %
%   N9:43  ADS_MANUAL  "STATE ADS Manual" %
%   N15:4/0  MAN_ADSA_REGEN_INOUT  "CONTROL Manually open the ADS A regen in and out valves" %
%   O:2.0/0  ADS_A_REGEN_IN_OUT  "SV-1" %
% Rung: 29 %
% If the state of this machine is REGEN and the regen process is calling for the heaters to operate, operate the heaters %
SOR BST XIC B38:0/2 NXB XIC B34:1/0 BND XIO B38:0/3 XIO B38:0/4 XIO B38:0/5 XIC B38:0/0 XIC B38:0/1 OTE B34:1/0 EOR
%   B38:0/2  MAN_ADS_A_HTRS_ON  "COMMAND HMI" %
%   B34:1/0  MAN_ADS_A_HTR_ON_EN %
%   B38:0/3  MAN_ADS_B_HTRS_ON  "COMMAND HMI" %
%   B38:0/4  MAN_ADS_C_HTRS_ON  "COMMAND HMI" %
%   B38:0/5  MAN_ADS_D_HTRS_ON  "COMMAND HMI" %
%   B38:0/0  MAN_HTR_OVERRIDE  "COMMAND HMI" %
%   B38:0/1  MAN_ADS_HTRS_ON  "COMMAND HMI" %

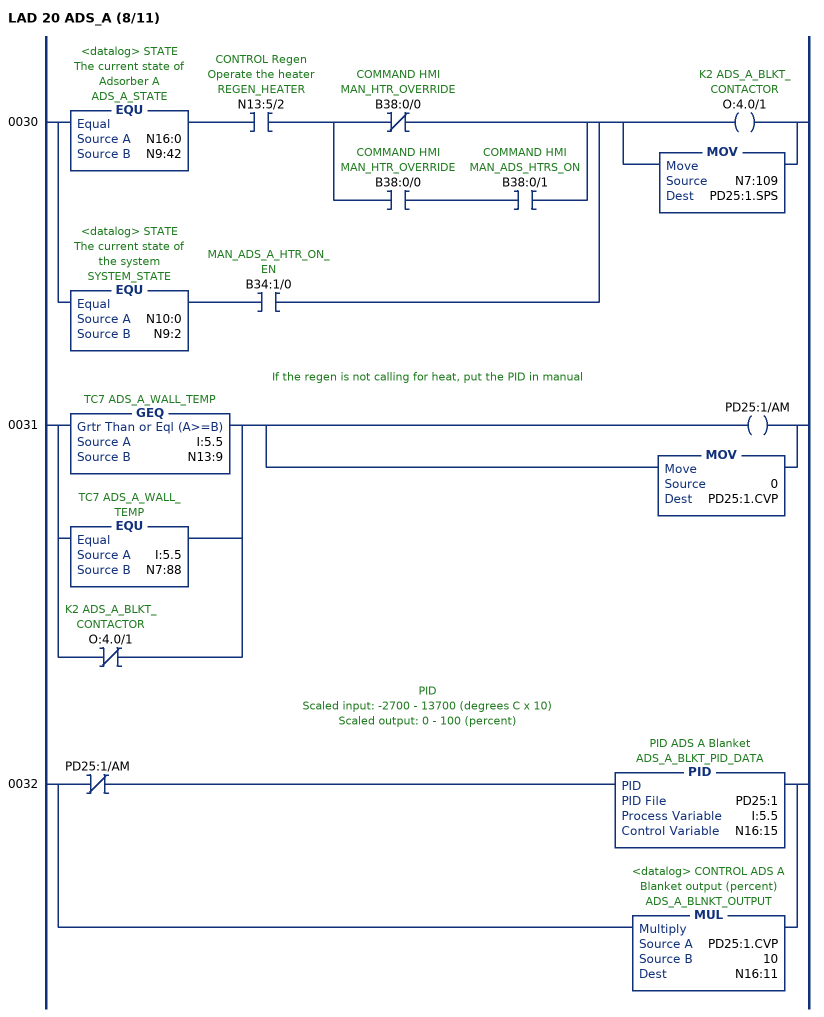
% Rung: 30 %
SOR BST EQU N16:0 N9:42 XIC N13:5/2 BST XIO B38:0/0 NXB XIC B38:0/0 XIC B38:0/1 BND NXB EQU N10:0 N9:2 XIC B34:1/0 BND BST OTE O:4.0/1 NXB MOV N7:109 PD25:1.SPS BND EOR
%   N16:0  ADS_A_STATE  "<datalog> STATE The current state of Adsorber A" %
%   N9:42  ADS_REGEN  "STATE ADS Regen" %
%   N13:5/2  REGEN_HEATER  "CONTROL Regen Operate the heater" %
%   B38:0/0  MAN_HTR_OVERRIDE  "COMMAND HMI" %
%   B38:0/1  MAN_ADS_HTRS_ON  "COMMAND HMI" %
%   N10:0  SYSTEM_STATE  "<datalog> STATE The current state of the system" %
%   N9:2  SYSTEM_MANUAL  "STATE System Manual" %
%   B34:1/0  MAN_ADS_A_HTR_ON_EN %
%   O:4.0/1  ADS_A_BLKT_CONTACTOR  "K2" %
%   N7:109  BLANKET_SP  "<datalog> ADS Blanket PID Setpoint" %
% Rung: 31 %
% If the regen is not calling for heat, put the PID in manual %
SOR BST GEQ I:5.5 N13:9 NXB EQU I:5.5 N7:88 NXB XIO O:4.0/1 BND BST OTE PD25:1/AM NXB MOV 0 PD25:1.CVP BND EOR
%   I:5.5  ADS_A_WALL_TEMP  "TC7" %
%   N13:9  BLANKET_LIMIT  "ADS Blanket Temp Limit" %
%   N7:88  TC_OPEN_SP  "CONFIG TC Open Setpoint" %
%   O:4.0/1  ADS_A_BLKT_CONTACTOR  "K2" %
% Rung: 32 %
% PID
% Scaled input: -2700 - 13700 (degrees C x 10)
% Scaled output: 0 - 100 (percent) %
SOR BST XIO PD25:1/AM PID PD25:1 I:5.5 N16:15 NXB MUL PD25:1.CVP 10 N16:11 BND EOR
%   PD25:1  ADS_A_BLKT_PID_DATA  "PID ADS A Blanket" %
%   I:5.5  ADS_A_WALL_TEMP  "TC7" %
%   N16:15  ADS_A_BLKT_OUTPT_RAW  "CONTROL ADS A Blanket PID Output Raw" %
%   N16:11  ADS_A_BLNKT_OUTPUT  "<datalog> CONTROL ADS A Blanket output (percent)" %

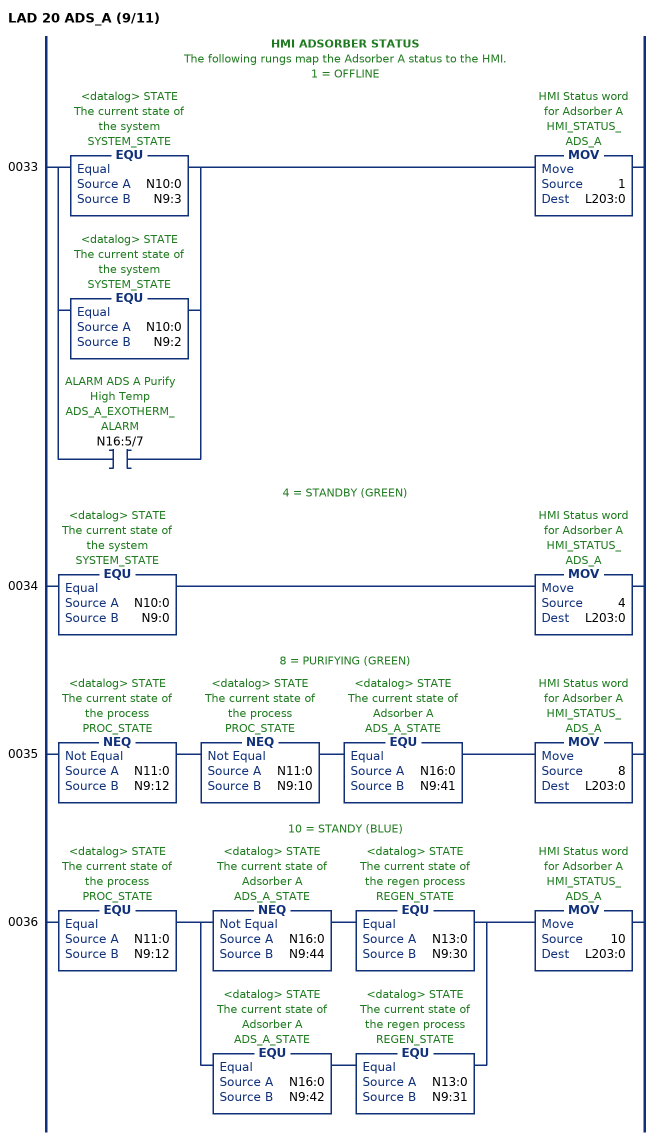
% Rung: 33 %
% TITLE: HMI ADSORBER STATUS %
% The following rungs map the Adsorber A status to the HMI.
% 1 = OFFLINE %
SOR BST EQU N10:0 N9:3 NXB EQU N10:0 N9:2 NXB XIC N16:5/7 BND MOV 1 L203:0 EOR
%   N10:0  SYSTEM_STATE  "<datalog> STATE The current state of the system" %
%   N9:3  SYSTEM_ALARM  "STATE System Alarm" %
%   N9:2  SYSTEM_MANUAL  "STATE System Manual" %
%   N16:5/7  ADS_A_EXOTHERM_ALARM  "ALARM ADS A Purify High Temp" %
%   L203:0  HMI_STATUS_ADS_A  "HMI Status word for Adsorber A" %
% Rung: 34 %
% 4 = STANDBY (GREEN) %
SOR EQU N10:0 N9:0 MOV 4 L203:0 EOR
%   N10:0  SYSTEM_STATE  "<datalog> STATE The current state of the system" %
%   N9:0  SYSTEM_STANDBY  "STATE System Standby" %
%   L203:0  HMI_STATUS_ADS_A  "HMI Status word for Adsorber A" %
% Rung: 35 %
% 8 = PURIFYING (GREEN) %
SOR NEQ N11:0 N9:12 NEQ N11:0 N9:10 EQU N16:0 N9:41 MOV 8 L203:0 EOR
%   N11:0  PROC_STATE  "<datalog> STATE The current state of the process" %
%   N9:12  PROC_REGEN_A  "STATE Process Regen A" %
%   N9:10  PROCESS_STANDBY  "STATE Process Standby" %
%   N16:0  ADS_A_STATE  "<datalog> STATE The current state of Adsorber A" %
%   N9:41  ADS_PURIFY  "STATE ADS Purify" %
%   L203:0  HMI_STATUS_ADS_A  "HMI Status word for Adsorber A" %
% Rung: 36 %
% 10 = STANDY (BLUE) %
SOR EQU N11:0 N9:12 BST NEQ N16:0 N9:44 EQU N13:0 N9:30 NXB EQU N16:0 N9:42 EQU N13:0 N9:31 BND MOV 10 L203:0 EOR
%   N11:0  PROC_STATE  "<datalog> STATE The current state of the process" %
%   N9:12  PROC_REGEN_A  "STATE Process Regen A" %
%   N16:0  ADS_A_STATE  "<datalog> STATE The current state of Adsorber A" %
%   N9:44  ADS_ALARM  "STATE ADS Alarm" %
%   N13:0  REGEN_STATE  "<datalog> STATE The current state of the regen process" %
%   N9:30  REGEN_STANDBY  "STATE Regen Standby" %
%   N9:42  ADS_REGEN  "STATE ADS Regen" %
%   N9:31  REGEN_DELAY  "STATE Regen Delay" %
%   L203:0  HMI_STATUS_ADS_A  "HMI Status word for Adsorber A" %

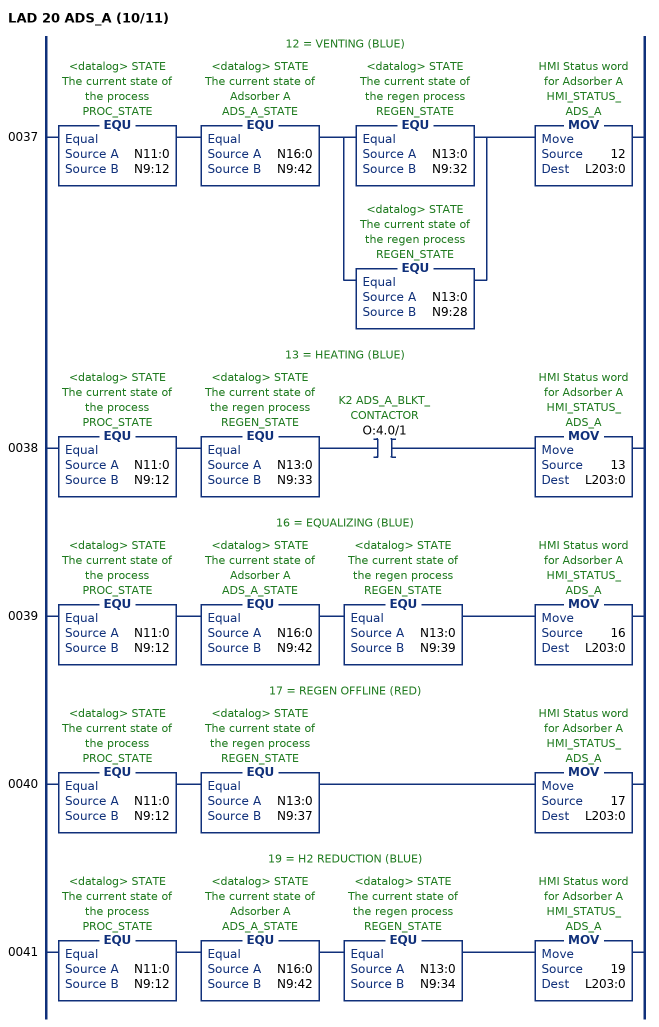
% Rung: 37 %
% 12 = VENTING (BLUE) %
SOR EQU N11:0 N9:12 EQU N16:0 N9:42 BST EQU N13:0 N9:32 NXB EQU N13:0 N9:28 BND MOV 12 L203:0 EOR
%   N11:0  PROC_STATE  "<datalog> STATE The current state of the process" %
%   N9:12  PROC_REGEN_A  "STATE Process Regen A" %
%   N16:0  ADS_A_STATE  "<datalog> STATE The current state of Adsorber A" %
%   N9:42  ADS_REGEN  "STATE ADS Regen" %
%   N13:0  REGEN_STATE  "<datalog> STATE The current state of the regen process" %
%   N9:32  REGEN_VENT  "STATE Regen Vent" %
%   N9:28  REGEN_VENT_2 %
%   L203:0  HMI_STATUS_ADS_A  "HMI Status word for Adsorber A" %
% Rung: 38 %
% 13 = HEATING (BLUE) %
SOR EQU N11:0 N9:12 EQU N13:0 N9:33 XIC O:4.0/1 MOV 13 L203:0 EOR
%   N11:0  PROC_STATE  "<datalog> STATE The current state of the process" %
%   N9:12  PROC_REGEN_A  "STATE Process Regen A" %
%   N13:0  REGEN_STATE  "<datalog> STATE The current state of the regen process" %
%   N9:33  REGEN_HEAT_BED  "STATE Regen Heat wall" %
%   O:4.0/1  ADS_A_BLKT_CONTACTOR  "K2" %
%   L203:0  HMI_STATUS_ADS_A  "HMI Status word for Adsorber A" %
% Rung: 39 %
% 16 = EQUALIZING (BLUE) %
SOR EQU N11:0 N9:12 EQU N16:0 N9:42 EQU N13:0 N9:39 MOV 16 L203:0 EOR
%   N11:0  PROC_STATE  "<datalog> STATE The current state of the process" %
%   N9:12  PROC_REGEN_A  "STATE Process Regen A" %
%   N16:0  ADS_A_STATE  "<datalog> STATE The current state of Adsorber A" %
%   N9:42  ADS_REGEN  "STATE ADS Regen" %
%   N13:0  REGEN_STATE  "<datalog> STATE The current state of the regen process" %
%   N9:39  REGEN_EQUALIZE  "STATE Regen Equalize" %
%   L203:0  HMI_STATUS_ADS_A  "HMI Status word for Adsorber A" %
% Rung: 40 %
% 17 = REGEN OFFLINE (RED) %
SOR EQU N11:0 N9:12 EQU N13:0 N9:37 MOV 17 L203:0 EOR
%   N11:0  PROC_STATE  "<datalog> STATE The current state of the process" %
%   N9:12  PROC_REGEN_A  "STATE Process Regen A" %
%   N13:0  REGEN_STATE  "<datalog> STATE The current state of the regen process" %
%   N9:37  REGEN_ALARM  "STATE Regen Alarm" %
%   L203:0  HMI_STATUS_ADS_A  "HMI Status word for Adsorber A" %
% Rung: 41 %
% 19 = H2 REDUCTION (BLUE) %
SOR EQU N11:0 N9:12 EQU N16:0 N9:42 EQU N13:0 N9:34 MOV 19 L203:0 EOR
%   N11:0  PROC_STATE  "<datalog> STATE The current state of the process" %
%   N9:12  PROC_REGEN_A  "STATE Process Regen A" %
%   N16:0  ADS_A_STATE  "<datalog> STATE The current state of Adsorber A" %
%   N9:42  ADS_REGEN  "STATE ADS Regen" %
%   N13:0  REGEN_STATE  "<datalog> STATE The current state of the regen process" %
%   N9:34  REGEN_H2_REDUCTION  "STATE Regen Running" %
%   L203:0  HMI_STATUS_ADS_A  "HMI Status word for Adsorber A" %

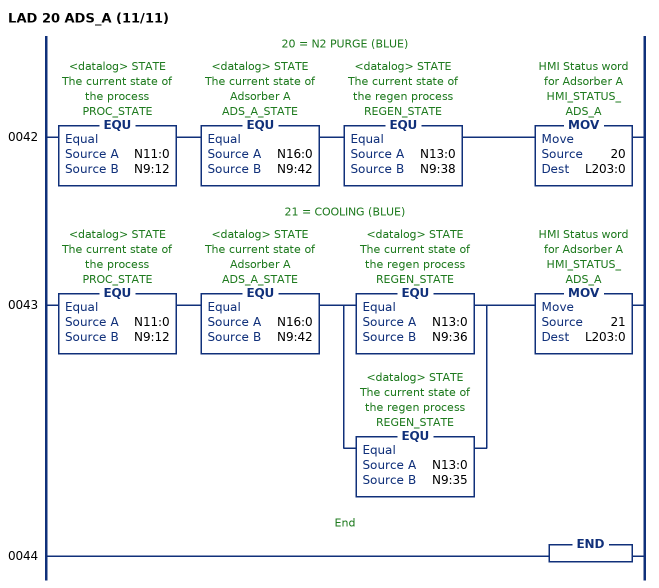
% Rung: 42 %
% 20 = N2 PURGE (BLUE) %
SOR EQU N11:0 N9:12 EQU N16:0 N9:42 EQU N13:0 N9:38 MOV 20 L203:0 EOR
%   N11:0  PROC_STATE  "<datalog> STATE The current state of the process" %
%   N9:12  PROC_REGEN_A  "STATE Process Regen A" %
%   N16:0  ADS_A_STATE  "<datalog> STATE The current state of Adsorber A" %
%   N9:42  ADS_REGEN  "STATE ADS Regen" %
%   N13:0  REGEN_STATE  "<datalog> STATE The current state of the regen process" %
%   N9:38  REGEN_PURGE  "STATE Regen Hot Purge" %
%   L203:0  HMI_STATUS_ADS_A  "HMI Status word for Adsorber A" %
% Rung: 43 %
% 21 = COOLING (BLUE) %
SOR EQU N11:0 N9:12 EQU N16:0 N9:42 BST EQU N13:0 N9:36 NXB EQU N13:0 N9:35 BND MOV 21 L203:0 EOR
%   N11:0  PROC_STATE  "<datalog> STATE The current state of the process" %
%   N9:12  PROC_REGEN_A  "STATE Process Regen A" %
%   N16:0  ADS_A_STATE  "<datalog> STATE The current state of Adsorber A" %
%   N9:42  ADS_REGEN  "STATE ADS Regen" %
%   N13:0  REGEN_STATE  "<datalog> STATE The current state of the regen process" %
%   N9:36  REGEN_COOL  "STATE Regen Cool" %
%   N9:35  REGEN_COOL_WALL  "STATE Regen Cool wall" %
%   L203:0  HMI_STATUS_ADS_A  "HMI Status word for Adsorber A" %
% Rung: 44 %
% End %
SOR END EOR

LADDER 21 "ADS_A_FLT"    % Controls the Adsorber A faults %
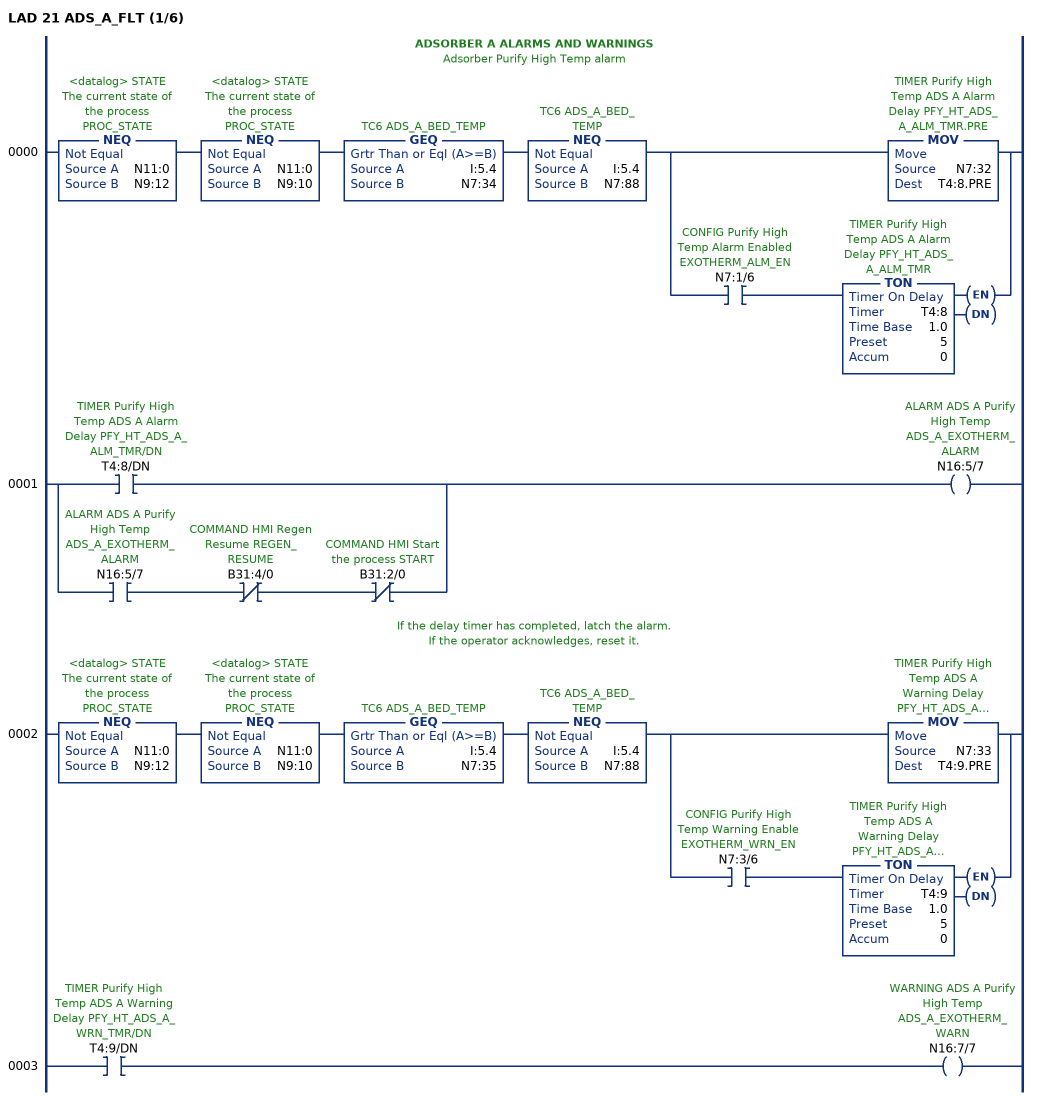
% Rung: 0 %
% TITLE: ADSORBER A ALARMS AND WARNINGS %
% Adsorber Purify High Temp alarm %
SOR NEQ N11:0 N9:12 NEQ N11:0 N9:10 GEQ I:5.4 N7:34 NEQ I:5.4 N7:88 BST MOV N7:32 T4:8.PRE NXB XIC N7:1/6 TON T4:8 1.0 5 0 BND EOR
%   N11:0  PROC_STATE  "<datalog> STATE The current state of the process" %
%   N9:12  PROC_REGEN_A  "STATE Process Regen A" %
%   N9:10  PROCESS_STANDBY  "STATE Process Standby" %
%   I:5.4  ADS_A_BED_TEMP  "TC6" %
%   N7:34  EXOTHERM_ALM_SP  "CONFIG Purify High Temp Alarm Setpoint" %
%   N7:88  TC_OPEN_SP  "CONFIG TC Open Setpoint" %
%   N7:32  EXOTHERM_ALM_DLY  "CONFIG Purify High Temp Alarm Delay" %
%   T4:8  PFY_HT_ADS_A_ALM_TMR  "TIMER Purify High Temp ADS A Alarm Delay" %
%   N7:1/6  EXOTHERM_ALM_EN  "CONFIG Purify High Temp Alarm Enabled" %
% Rung: 1 %
SOR BST XIC T4:8/DN NXB XIC N16:5/7 XIO B31:4/0 XIO B31:2/0 BND OTE N16:5/7 EOR
%   T4:8  PFY_HT_ADS_A_ALM_TMR  "TIMER Purify High Temp ADS A Alarm Delay" %
%   N16:5/7  ADS_A_EXOTHERM_ALARM  "ALARM ADS A Purify High Temp" %
%   B31:4/0  REGEN_RESUME  "COMMAND HMI Regen Resume" %
%   B31:2/0  START  "COMMAND HMI Start the process" %
% Rung: 2 %
% If the delay timer has completed, latch the alarm.
% If the operator acknowledges, reset it. %
SOR NEQ N11:0 N9:12 NEQ N11:0 N9:10 GEQ I:5.4 N7:35 NEQ I:5.4 N7:88 BST MOV N7:33 T4:9.PRE NXB XIC N7:3/6 TON T4:9 1.0 5 0 BND EOR
%   N11:0  PROC_STATE  "<datalog> STATE The current state of the process" %
%   N9:12  PROC_REGEN_A  "STATE Process Regen A" %
%   N9:10  PROCESS_STANDBY  "STATE Process Standby" %
%   I:5.4  ADS_A_BED_TEMP  "TC6" %
%   N7:35  EXOTHERM_WRN_SP  "CONFIG Purify High Temp Warning Setpoint" %
%   N7:88  TC_OPEN_SP  "CONFIG TC Open Setpoint" %
%   N7:33  EXOTHERM_WRN_DLY  "CONFIG Purify High Temp Warning Delay" %
%   T4:9  PFY_HT_ADS_A_WRN_TMR  "TIMER Purify High Temp ADS A Warning Delay" %
%   N7:3/6  EXOTHERM_WRN_EN  "CONFIG Purify High Temp Warning Enable" %
% Rung: 3 %
SOR XIC T4:9/DN OTE N16:7/7 EOR
%   T4:9  PFY_HT_ADS_A_WRN_TMR  "TIMER Purify High Temp ADS A Warning Delay" %
%   N16:7/7  ADS_A_EXOTHERM_WARN  "WARNING ADS A Purify High Temp" %

